// ---- 20_Product/20_ProBox/30_Toolbox/F_AssignTU_DataIndexToZone.TcPOU
FUNCTION F_AssignTU_DataIndexToZone : BOOL
(**************************************************************************************
 * 	Application		:	BoxControl Framework
 *	Revision		:	$Revision: $
 *	Revision date	:	$Date: $
 *	Last changed by	:	$Author: q8sheds $
 *	URL				:	$URL: $
 *
 *	Purpose			:	assign TU data to zone, overrides former method M_AssignTU_DataIndexToZone
 *
 * ------------------------------------------------------------------------------------
 *	Copyright Swisslog [IP AG], Switzerland. All rights reserved.
 * 
 * ------------------------------------------------------------------------------------
 *	
 * 	Revision History: 
 *
 * 	VERSION			DATE			INITIALS			DESCRIPTION
 *	0.1				2018-05-31		PkF/RtK					First Version
 *
 **************************************************************************************)
VAR_INPUT
	eFunctionNumber		: E_FunctionNumber;
	ZoneNumber			: INT; 
	TU_DataIndex		: DINT;
END_VAR

F_AssignTU_DataIndexToZone := FALSE;

// Check if function number and zone is valid
IF eFunctionNumber > E_FunctionNumber.F_BEGIN_FUNCTION AND
   eFunctionNumber < E_FunctionNumber.F_END_FUNCTION AND
   ZoneNumber > 0 AND ZoneNumber <= NUMBER_OF_ZONES_PER_FUNCTION THEN
  
   // yes, Zone number is valid	
	// Check reference is valid
    IF( NOT __ISVALIDREF(FunctionRegistry[eFunctionNumber].rFunction) OR
		NOT __ISVALIDREF(FunctionRegistry[eFunctionNumber].rSettingsFunction) OR
		NOT __ISVALIDREF(FunctionRegistry[eFunctionNumber].Zone[ZoneNumber].refZoneData)) THEN
		RETURN;  //bad references
	END_IF		
   
	
	IF ZoneNumber > 0 AND ZoneNumber <= FunctionRegistry[eFunctionNumber].rSettingsFunction.NumberOfZones THEN
		// TU Index is equal to the current
		IF TU_DataIndex > 0 AND FunctionRegistry[eFunctionNumber].Zone[ZoneNumber].refZoneData.TransportControlData.TU_DataIndex = 0 THEN
			// Assign TU data index						
			FunctionRegistry[eFunctionNumber].Zone[ZoneNumber].refZoneData.TransportControlData.TU_DataIndex := TU_DataIndex;
			//LastTU_DataIndex is not changed.
			FunctionRegistry[eFunctionNumber].Zone[ZoneNumber].refZoneData.TransportControlData.DataPresent := TRUE;
			F_AssignTU_DataIndexToZone := TRUE; 
		END_IF
	END_IF	   
      
END_IF

END_FUNCTION

// ---- 20_Product/20_ProBox/30_Toolbox/F_CheckAllFree.TcPOU
FUNCTION F_CheckAllFree : BOOL
(**************************************************************************************
 * 	Application		:	BoxControl Framework
 *	Revision		:	$Revision: 417092 $
 *	Revision date	:	$Date: 2018-11-14 12:58:58 +0100 (Mi., 14 Nov 2018) $
 *	Last changed by	:	$Author: q8aberh $
 *	URL				:	$URL: http://almscdc.swisslog.com/repo/SWPD/Development/ProMove/02_Controls/ProBox/03_Implementation/01_DevelopmentProject/01_Software/ProBox_COE/ProBox_DevProj_v1.0/PLC_1/20_Product/10_App/12_E_Functions/11_ProBox/02_Functions/02_TransportControl/F_Che $
 *
 *	Purpose			:	Return number of zones
 *
 * ------------------------------------------------------------------------------------
 *	Copyright Swisslog [IP AG], Switzerland. All rights reserved.
 * 
 * ------------------------------------------------------------------------------------
 *	
 * 	Revision History: 
 *
 * 	VERSION			DATE			INITIALS			DESCRIPTION
 *	0.1				01.01.2001		swl					Example
 *
 **************************************************************************************)
VAR_INPUT
	eFunctionNumber		: E_FunctionNumber; // Function number
END_VAR
VAR
	idx 				: INT; // Iterator
	AllFree				: BOOL; // Temp to check if all zones are occupied
END_VAR

// Check if function number is valid
IF eFunctionNumber > E_FunctionNumber.F_BEGIN_FUNCTION AND
   eFunctionNumber < E_FunctionNumber.F_END_FUNCTION THEN
  
   // Check reference is valid
   IF __ISVALIDREF(FunctionRegistry[eFunctionNumber].rSettingsFunction) THEN
		// Return All Free
		AllFree := TRUE;
		FOR idx := 1 TO FunctionRegistry[eFunctionNumber].rSettingsFunction.NumberOfZones DO
			IF FunctionRegistry[eFunctionNumber].Zone[idx].refZoneData.TransportControlData.Occupied THEN
				AllFree := FALSE;
				EXIT;
			END_IF
		END_FOR
		F_CheckAllFree := AllFree;
   END_IF
END_IF

END_FUNCTION

// ---- 20_Product/20_ProBox/30_Toolbox/F_CheckAllOccupied.TcPOU
FUNCTION F_CheckAllOccupied : BOOL
(**************************************************************************************
 * 	Application		:	BoxControl Framework
 *	Revision		:	$Revision: 417092 $
 *	Revision date	:	$Date: 2018-11-14 12:58:58 +0100 (Mi., 14 Nov 2018) $
 *	Last changed by	:	$Author: q8aberh $
 *	URL				:	$URL: http://almscdc.swisslog.com/repo/SWPD/Development/ProMove/02_Controls/ProBox/03_Implementation/01_DevelopmentProject/01_Software/ProBox_COE/ProBox_DevProj_v1.0/PLC_1/20_Product/10_App/12_E_Functions/11_ProBox/02_Functions/02_TransportControl/F_Che $
 *
 *	Purpose			:	Return number of zones
 *
 * ------------------------------------------------------------------------------------
 *	Copyright Swisslog [IP AG], Switzerland. All rights reserved.
 * 
 * ------------------------------------------------------------------------------------
 *	
 * 	Revision History: 
 *
 * 	VERSION			DATE			INITIALS			DESCRIPTION
 *	0.1				01.01.2001		swl					Example
 *
 **************************************************************************************)
VAR_INPUT
	eFunctionNumber		: E_FunctionNumber; // Function number
END_VAR
VAR
	idx 				: INT; // Iterator
	AllOccupied			: BOOL; // Temp to check if all zones are free
END_VAR

// Check if function number is valid
IF eFunctionNumber > E_FunctionNumber.F_BEGIN_FUNCTION AND
   eFunctionNumber < E_FunctionNumber.F_END_FUNCTION THEN
  
   // Check reference is valid
   IF __ISVALIDREF(FunctionRegistry[eFunctionNumber].rSettingsFunction) THEN
		// Return All Occupied
		AllOccupied := TRUE;
		FOR idx := 1 TO FunctionRegistry[eFunctionNumber].rSettingsFunction.NumberOfZones DO
			IF NOT FunctionRegistry[eFunctionNumber].Zone[idx].refZoneData.TransportControlData.Occupied THEN
				AllOccupied := FALSE;
				EXIT;
			END_IF
		END_FOR
		F_CheckAllOccupied := AllOccupied;
   END_IF
END_IF

END_FUNCTION

// ---- 20_Product/20_ProBox/30_Toolbox/F_CheckAllStarted.TcPOU
FUNCTION F_CheckAllStarted : BOOL
(**************************************************************************************
 * 	Application		:	BoxControl Framework
 *	Revision		:	$Revision: 417092 $
 *	Revision date	:	$Date: 2018-11-14 12:58:58 +0100 (Mi., 14 Nov 2018) $
 *	Last changed by	:	$Author: q8aberh $
 *	URL				:	$URL: http://almscdc.swisslog.com/repo/SWPD/Development/ProMove/02_Controls/ProBox/03_Implementation/01_DevelopmentProject/01_Software/ProBox_COE/ProBox_DevProj_v1.0/PLC_1/20_Product/10_App/12_E_Functions/11_ProBox/02_Functions/02_TransportControl/F_Che $
 *
 *	Purpose			:	Returns true if all the zones on the function are started
 *
 * ------------------------------------------------------------------------------------
 *	Copyright Swisslog [IP AG], Switzerland. All rights reserved.
 * 
 * ------------------------------------------------------------------------------------
 *	
 * 	Revision History: 
 *
 * 	VERSION			DATE			INITIALS			DESCRIPTION
 *	0.1				2018-08-14		PkF					First version
 *
 **************************************************************************************)
VAR_INPUT
	eFunctionNumber		: E_FunctionNumber; // Function number
END_VAR
VAR
	idx 				: INT; // Iterator
	AllStarted			: BOOL; // Temp to check if all zones are started
END_VAR

// Check if function number is valid
IF eFunctionNumber > E_FunctionNumber.F_BEGIN_FUNCTION AND
   eFunctionNumber < E_FunctionNumber.F_END_FUNCTION THEN
  
   // Check reference is valid
   IF __ISVALIDREF(FunctionRegistry[eFunctionNumber].rSettingsFunction) AND 
		__ISVALIDREF(FunctionRegistry[eFunctionNumber].rFunctionData) THEN
		// Return All Started
		AllStarted := TRUE;
		FOR idx := 1 TO FunctionRegistry[eFunctionNumber].rSettingsFunction.NumberOfZones DO
			IF (FunctionRegistry[eFunctionNumber].rFunctionData.OperationState.eState <> E_PositionState.STARTED AND 
				FunctionRegistry[eFunctionNumber].rFunctionData.OperationState.eState <> E_PositionState.STOPPING) OR 
				FunctionRegistry[eFunctionNumber].rFunctionData.ErrorData.ZoneErrorPending THEN
				AllStarted := FALSE;
				EXIT;
			END_IF
		END_FOR
		F_CheckAllStarted := AllStarted;
   END_IF
END_IF

END_FUNCTION

// ---- 20_Product/20_ProBox/30_Toolbox/F_DeleteTU_DataIndex.TcPOU
FUNCTION F_DeleteTU_DataIndex : BOOL
(**************************************************************************************
 * 	Application		:	BoxControl Framework
 *	Revision		:	$Revision: 417092 $
 *	Revision date	:	$Date: 2018-11-14 12:58:58 +0100 (Mi., 14 Nov 2018) $
 *	Last changed by	:	$Author: q8aberh $
 *	URL				:	$URL: http://almscdc.swisslog.com/repo/SWPD/Development/ProMove/02_Controls/ProBox/03_Implementation/01_DevelopmentProject/01_Software/ProBox_COE/ProBox_DevProj_v1.0/PLC_1/20_Product/10_App/12_E_Functions/11_ProBox/02_Functions/F_DeleteTU_DataIndex.TcPO $
 *
 *	Purpose			:	Moves TU data from a position.
 *
 * ------------------------------------------------------------------------------------
 *	Copyright Swisslog [IP AG], Switzerland. All rights reserved.
 * 
 * ------------------------------------------------------------------------------------
 *	
 * 	Revision History: 
 *
 * 	VERSION			DATE			INITIALS			DESCRIPTION
 *	0.1				01.01.2001		swl					Example
 *
 **************************************************************************************)
VAR_INPUT
	eFunctionNumber	: E_FunctionNumber; // Function number of corresponding function
	mZoneNumber 	: INT; // Zone number
END_VAR

VAR
	STI_Instance	: ITF_SubsystemTransport; // Instance to compare valid interfaces
END_VAR

// Check if function number is valid
IF eFunctionNumber > E_FunctionNumber.F_BEGIN_FUNCTION AND
   eFunctionNumber < E_FunctionNumber.F_END_FUNCTION THEN
  
	// Check reference is valid
	IF __ISVALIDREF(FunctionRegistry[eFunctionNumber].rFunction) THEN
   		// Return tu data index
   		F_DeleteTU_DataIndex := FunctionRegistry[eFunctionNumber].rFunction.M_DeleteTU_DataIndex(
						mZoneNumber := mZoneNumber,
						mTU_DataIndex := F_GetTU_DataIndex(
												eFunctionNumber := eFunctionNumber,
												ZoneNumber := mZoneNumber),
						mInit	:= FALSE);
	END_IF
END_IF

END_FUNCTION

// ---- 20_Product/20_ProBox/30_Toolbox/F_PB_GetTransportData.TcPOU
FUNCTION F_PB_GetTransportData : ST_TransportData
(**************************************************************************************
 * 	Application		:	BoxControl Framework
 *	Revision		:	$Revision:  $
 *	Revision date	:	$Date: $
 *	Last changed by	:	$Author: q8sheds $
 *	URL				:	$URL: $
 *
 *	Purpose			:	return Transport data
 *
 * ------------------------------------------------------------------------------------
 *	Copyright Swisslog [IP AG], Switzerland. All rights reserved.
 * 
 * ------------------------------------------------------------------------------------
 *	
 * 	Revision History: 
 *
 * 	VERSION			DATE			INITIALS			DESCRIPTION
 *	0.1				01.01.2001		swl					Example
 *
 **************************************************************************************)
VAR_INPUT
	eFunctionNumber		: E_FunctionNumber; // Function number
	ZoneNumber			: INT; // Zone number
END_VAR



VAR
	FunctionBase: INT;
END_VAR


//init default data
F_PB_GetTransportData.eFunctionNumber := E_FunctionNumber.F_BEGIN_FUNCTION;
F_PB_GetTransportData.ZoneNumber:=0;
F_PB_GetTransportData.rTransportControlData REF= PBTransportCtrl.pbTransportControlDataEmpty;
F_PB_GetTransportData.rSettings REF= PBTransportCtrl.pbZoneSettingsEmpty;


// Check if function number is valid
IF eFunctionNumber > E_FunctionNumber.F_BEGIN_FUNCTION AND
   eFunctionNumber < E_FunctionNumber.F_END_FUNCTION AND
   ZoneNumber > 0 AND ZoneNumber <= NUMBER_OF_ZONES_PER_FUNCTION THEN
  
	// Check reference is valid
	IF __ISVALIDREF(FunctionRegistry[eFunctionNumber].Zone[ZoneNumber].refZoneData) THEN
   		// Set transport data
   		//F_PB_GetTransportControlDataRef REF= FunctionRegistry[eFunctionNumber].Zone[ZoneNumber].refZoneData.TransportControlData;
		F_PB_GetTransportData.eFunctionNumber := eFunctionNumber;
		F_PB_GetTransportData.ZoneNumber := ZoneNumber;
		F_PB_GetTransportData.rSettings REF= FunctionRegistry[eFunctionNumber].rSettingsFunction.Zone[ZoneNumber];
		F_PB_GetTransportData.rTransportControlData REF= FunctionRegistry[eFunctionNumber].Zone[ZoneNumber].refZoneData.TransportControlData;				
	END_IF
END_IF

END_FUNCTION

// ---- 20_Product/20_ProBox/30_Toolbox/F_PB_GetZoneITC.TcPOU
FUNCTION F_PB_GetZoneITC : ST_ITC_Zone
VAR_INPUT
		eFunctionNumber		: E_FunctionNumber; // Function number
		ZoneNumber			: INT := 1;
END_VAR
VAR
END_VAR

// Check if function number is validas
IF eFunctionNumber > E_FunctionNumber.F_BEGIN_FUNCTION AND
   eFunctionNumber < E_FunctionNumber.F_END_FUNCTION THEN
  
	// Check reference is valid
	IF __ISVALIDREF(FunctionRegistry[eFunctionNumber].rFunctionInterface) THEN
   		// Return function interlock
   		F_PB_GetZoneITC := FunctionRegistry[eFunctionNumber].rFunction.ITC.ZoneITC[ZoneNumber];
	END_IF
END_IF

END_FUNCTION

// ---- 20_Product/20_ProBox/30_Toolbox/F_PB_IsLogicalOccupied.TcPOU
//A zone is occupied until the TU is handed over completly, or when the takeover is fully completed
FUNCTION F_PB_IsLogicalOccupied : BOOL
VAR_INPUT
	TransportControlData : REFERENCE TO ST_TransportControlData;
END_VAR
VAR
END_VAR


IF(NOT __ISVALIDREF(TransportControlData)) THEN RETURN; END_IF;

F_PB_IsLogicalOccupied := TransportControlData.Occupied OR TransportControlData.eTransportState = E_TransportState.HANDOVER;

END_FUNCTION

// ---- 20_Product/20_ProBox/30_Toolbox/F_PB_SetDestination.TcPOU
//Set destination to an already existing TU Table dataset
FUNCTION F_PB_SetDestination : BOOL
(**************************************************************************************
 * 	Application		:	ProBox
 *	Revision		:	$$
 *	Revision date	:	$$
 *	Last changed by	:	$$
 *	URL				:	$$
 *
 *	Purpose			:	Set a destination to an existing TU Table dataset.
 * 						Remark: as Tu_Table is persistant memory type, one should not repeatedly write to the TU_Table 
 *
 * ------------------------------------------------------------------------------------
 *	Copyright Swisslog [IP AG], Switzerland. All rights reserved.  
 **************************************************************************************)
VAR_INPUT
	TuDataIndex			: DINT; // Existing TU data table index there the Destination shall be assigned to
	Destination			: E_FunctionNumber; // Destination function
	DestinationZone		: INT:=1; // Destination zone
	ForceOverwrite		: BOOL:=FALSE; //Set to true in order to overwrite an existing valid destination and to be sure only writing once.
	AssignTuType		: BOOL:=FALSE; //Set to true to assign TuType
	TuType				: INT:=0;
	InsertFunction		: E_FunctionNumber:= E_FunctionNumber.F_BEGIN_FUNCTION;	//Optional data that is written to TimeStamp 
	InsertZone			: INT:=0;		
END_VAR
VAR
	DataSetDestIndex	: INT:=1;
END_VAR

//Sanity check
IF( TuDataIndex<=0 OR TuDataIndex>Conveyor.NUMBER_OF_TU_DATA OR
	Destination<= E_FunctionNumber.F_BEGIN_FUNCTION OR Destination>= E_FunctionNumber.F_END_FUNCTION OR
	DestinationZone <=0 OR DestinationZone > Conveyor.NUMBER_OF_ZONES_PER_FUNCTION) THEN
	RETURN; //invalid arguments
END_IF

IF(ForceOverwrite = FALSE AND TU_DataTable[TuDataIndex].DataSet.JobPresent) THEN
	RETURN; //JobPresent is active, so dont overwrite data again..
END_IF 


// Update TU Data set
TU_DataTable[TuDataIndex].DataSet.DataPresent:= TRUE;
TU_DataTable[TuDataIndex].DataSet.NumberOfDest	:= 1;				
TU_DataTable[TuDataIndex].DataSet.JobPresent := Destination > E_FunctionNumber.F_BEGIN_FUNCTION AND Destination<>InsertFunction;
TU_DataTable[TuDataIndex].Destination[DataSetDestIndex].eFunctionNumber := Destination;
TU_DataTable[TuDataIndex].Destination[DataSetDestIndex].ZoneNumber := DestinationZone;
TU_DataTable[TuDataIndex].Destination[DataSetDestIndex].PositionName := FunctionRegistry[Destination].FunctionName;

//Update TimeStamp
TU_DataTable[TuDataIndex].TimeStamp.eInsertFunctionNumber := InsertFunction;
TU_DataTable[TuDataIndex].TimeStamp.InsertZoneNumber:=InsertZone;
TU_DataTable[TuDataIndex].TimeStamp.InsertDateTime := System.fbSystemTime.TIMESTR;

//Set TU_Type?
IF(AssignTuType) THEN
	TU_DataTable[TuDataIndex].DataSet.TU_Type := TuType;
END_IF;


F_PB_SetDestination := TRUE;

END_FUNCTION

// ---- 20_Product/20_ProBox/30_Toolbox/F_PB_SetPalletOrientation.TcPOU
//Rotate profile data 90,80 or 270 degrees
FUNCTION F_PB_SetPalletOrientation : BOOL
VAR_INPUT
	ePalletOrientation  : E_PalletOrientation;	
	TuTableIdx			: DINT; // Which Tu Table destination slot (Default 1)
END_VAR
VAR
	TU_DataIndex  : DINT;
	_ProfileData: ST_Profile;
	_TempProfileData : ST_Profile;
	InvertedDone : BOOL:= FALSE;
END_VAR

//Sanity check
IF TuTableIdx <= 0 OR ePalletOrientation = OrientationZero THEN	
	RETURN;
END_IF

TU_DataIndex := TuTableIdx;
_ProfileData:= TU_DataTable[TU_DataIndex].Profile;	


CASE ePalletOrientation OF 	
	OrientationZero:
		; //nothing to do	

	OrientationNinty:
		TU_DataTable[TU_DataIndex].Profile.ProfileLeft:= _ProfileData.ProfileRear;	
		TU_DataTable[TU_DataIndex].Profile.ProfileRight:= _ProfileData.ProfileFront;	
		TU_DataTable[TU_DataIndex].Profile.ProfileFront:= _ProfileData.ProfileLeft;
		TU_DataTable[TU_DataIndex].Profile.ProfileRear:= _ProfileData.ProfileRight;
	
	OrientationOneEighty:
		TU_DataTable[TU_DataIndex].Profile.ProfileLeft:= _ProfileData.ProfileRight;
		TU_DataTable[TU_DataIndex].Profile.ProfileRight:= _ProfileData.ProfileLeft;
		TU_DataTable[TU_DataIndex].Profile.ProfileFront:= _ProfileData.ProfileRear;
		TU_DataTable[TU_DataIndex].Profile.ProfileRear:= _ProfileData.ProfileFront;
	
	OrientationTwoSeventy:
		TU_DataTable[TU_DataIndex].Profile.ProfileLeft:= _ProfileData.ProfileFront;
		TU_DataTable[TU_DataIndex].Profile.ProfileRight:= _ProfileData.ProfileRear;
		TU_DataTable[TU_DataIndex].Profile.ProfileFront:= _ProfileData.ProfileRight;
		TU_DataTable[TU_DataIndex].Profile.ProfileRear:= _ProfileData.ProfileLeft;
END_CASE

F_PB_SetPalletOrientation:=TRUE; ;

END_FUNCTION

// ---- 20_Product/20_ProBox/30_Toolbox/F_SetOccupied.TcPOU
FUNCTION F_SetOccupied : BOOL
(**************************************************************************************
 * 	Application		:	BoxControl Framework
 *	Revision		:	$Revision: 417092 $
 *	Revision date	:	$Date: 2018-11-14 12:58:58 +0100 (Mi., 14 Nov 2018) $
 *	Last changed by	:	$Author: q8aberh $
 *	URL				:	$URL: http://almscdc.swisslog.com/repo/SWPD/Development/ProMove/02_Controls/ProBox/03_Implementation/01_DevelopmentProject/01_Software/ProBox_COE/ProBox_DevProj_v1.0/PLC_1/20_Product/10_App/12_E_Functions/11_ProBox/02_Functions/F_SetOccupied.TcPOU $
 *
 *	Purpose			:	Return zone data
 *
 * ------------------------------------------------------------------------------------
 *	Copyright Swisslog [IP AG], Switzerland. All rights reserved.
 * 
 * ------------------------------------------------------------------------------------
 *	
 * 	Revision History: 
 *
 * 	VERSION			DATE			INITIALS			DESCRIPTION
 *	0.1				01.01.2001		swl					Example
 *
 **************************************************************************************)
VAR_INPUT
	eFunctionNumber		: E_FunctionNumber;
	ZoneNumber			: INT; 
END_VAR



// Check if function number and zone is valid
IF eFunctionNumber > E_FunctionNumber.F_BEGIN_FUNCTION AND
   eFunctionNumber < E_FunctionNumber.F_END_FUNCTION AND
   ZoneNumber > 0 AND ZoneNumber <= NUMBER_OF_ZONES_PER_FUNCTION THEN
  
	// Check reference is valid
    IF __ISVALIDREF(FunctionRegistry[eFunctionNumber].rFunction) THEN
	   // Return zone data
		IF __ISVALIDREF(FunctionRegistry[eFunctionNumber].Zone[ZoneNumber].refZoneData) THEN
			FunctionRegistry[eFunctionNumber].Zone[ZoneNumber].refZoneData.TransportControlData.Occupied := TRUE;
			FunctionRegistry[eFunctionNumber].Zone[ZoneNumber].refZoneData.TransportControlData.NumberOfPresentTUs :=1;
			FunctionRegistry[eFunctionNumber].Zone[ZoneNumber].refZoneData.TransportControlData.eTransportState := E_TransportState.OCCUPIED;
			F_SetOccupied:=TRUE;
	   END_IF
	    	   
    END_IF  
END_IF

END_FUNCTION

// ---- 20_Product/20_ProBox/40_TC_Visualization/99_SIS/FB_VizuSIS.TcPOU
FUNCTION_BLOCK FB_VizuSIS
VAR_INPUT
	ATQ				: BOOL;
	RTQ				: BOOL;
	TTA				: BOOL;
	TDQ				: BOOL;
	TTA_Destination	: STRING(NAME_LENGTH) := '10-001-0100-01-1';
	PositionString	: STRING(NAME_LENGTH) := '10-001-0100-01-1'; // Name of position 11-111-1111-11-1;	
	ATQ_Dimension	: ST_Dimension :=(Width:=800, Length:=800, Height:=500, Weight:=1200);
	ATQ_Label		: STRING(Conveyor.LABEL_LENGTH) := 'CREATECODE';
	TU_ID			: STRING(Conveyor.TU_ID_STRINGLENGTH):= Conveyor.TU_ID_UNKNOWN; // TU-ID
	AssignmentID	: UDINT := Conveyor.ASSIGNMENT_ID_UNKNOWN;
	AutoID			: BOOL; //Use TU ID and Assignment ID from TU table for TTA and TDQ
END_VAR
VAR_OUTPUT
	BadPosition		: BOOL;
END_VAR
VAR
	myPos			: STRING(NAME_LENGTH);
	myTuIndex		: DINT;

	TrigATQ : R_TRIG();
	TrigRTQ : R_TRIG();
	TrigTTA : R_TRIG();
	TrigTDQ : R_TRIG();
	
END_VAR
VAR_TEMP
	Position : ST_PositionIdent;
END_VAR

myPos := F_ReduceToAlphaNumeric(PositionString);
Position := F_SearchFunctionPosition(Position := myPos);
BadPosition := Position.eFunctionNumber = E_FunctionNumber.F_BEGIN_FUNCTION;
IF(BadPosition) THEN
	RETURN;
END_IF


TrigATQ(CLK:=ATQ);
TrigRTQ(CLK:=RTQ);
TrigTTA(CLK:=TTA);
TrigTDQ(CLK:=TDQ);

IF(TrigATQ.Q) THEN
	//ATQDimension
	_M_SendATQ(Position,ATQ_Dimension,ATQ_Label);
	//F_AddPhysicalTU(Position.eFunctionNumber,Position.ZoneNumber);
END_IF

IF(TrigRTQ.Q) THEN
	F_RemovePhysicalTU(Position.eFunctionNumber,Position.ZoneNumber);
END_IF

IF(TrigTTA.Q) THEN	
	_M_SendTTA(Position,TTA_Destination,TU_ID,AssignmentID);
END_IF

IF(TrigTDQ.Q) THEN	
	_M_SendTDQ(Position);
END_IF

METHOD PRIVATE _M_GetIDs : BOOL
VAR_INPUT
	Position 		: REFERENCE TO ST_PositionIdent;	
	TU_ID			: REFERENCE TO STRING(Conveyor.TU_ID_STRINGLENGTH); // TU-ID
	AssigID			: REFERENCE TO UDINT ;
END_VAR

VAR
	myTuIndex		: DINT;
END_VAR
//(Conveyor.TU_ID_STRINGLENGTH):= Conveyor.TU_ID_UNKNOWN;
//:= Conveyor.ASSIGNMENT_ID_UNKNOWN

IF(THIS^.AutoID) THEN
	
	myTuIndex := F_PB_GetTransportControlDataRef(Position.eFunctionNumber,Position.ZoneNumber).TU_DataIndex;
	IF(myTuIndex>0) THEN
		AssigID		:= TU_Table.TU_DataTable[myTuIndex].AssignmentID;
		TU_ID 			:= TU_Table.TU_DataTable[myTuIndex].TU_ID.ASCII;
	ELSE
		AssigID 		:= Conveyor.ASSIGNMENT_ID_UNKNOWN;
		TU_ID		:= Conveyor.TU_ID_UNKNOWN;	
	END_IF	
ELSE
	//use the ID's from the input field of the vizio interface.
	TU_ID := THIS^.TU_ID;	
	AssigID := THIS^.AssignmentID;
END_IF
END_METHOD

METHOD PRIVATE _M_SendATQ : BOOL
VAR_INPUT
	Position 		: REFERENCE TO ST_PositionIdent;
	Dimension		: REFERENCE TO ST_Dimension;
	Label			: REFERENCE TO STRING(Conveyor.LABEL_LENGTH);	
END_VAR
VAR
	myLabel			: STRING(Conveyor.LABEL_LENGTH);
END_VAR
VAR_STAT
	ID		: INT := 1;
	ATQ		: ST_ITC_ATQ;
END_VAR

ATQ.Position := F_ReduceToAlphaNumeric(InputString := Position.PositionName);

IF(Label[0]=0) THEN

	myLabel := F_StuffString(
			InputString 	:= INT_TO_STRING(ID), 
			StringLength	:= 8, 
			StuffCharacter 	:= '0',
			LeftAligned     := FALSE);
	myLabel := CONCAT('TESTLABEL_',myLabel);
			
	ID := ID + 1;
	IF ID > 9998 THEN
		ID := 1;
	END_IF
ELSE
	myLabel := Label;
END_IF		

IF(Dimension.Height=0) THEN Dimension.Height:=200; END_IF
IF(Dimension.Length=0) THEN Dimension.Length:=200; END_IF
IF(Dimension.Weight=0) THEN Dimension.Weight:=200; END_IF
IF(Dimension.Width=0) THEN Dimension.Width:=200; END_IF

ATQ.Height := Dimension.Height;
ATQ.Length := Dimension.Length;
ATQ.Weight := Dimension.Weight;
ATQ.Width := Dimension.Width;

ATQ.LabelPresent := 1;
ATQ.Label := myLabel;


IF(ProBoxSystem.EMULATION_ENABLED) THEN
	fbITC_ManagerEmulation.M_AddData(
		meChannelSrc := 0,
		mMsgType     := E_ITC_MsgTypeConv.E_ADD_TU_REQUEST,
		mpData		 := ADR(ATQ),
		mLen 		 := SIZEOF(ATQ));
END_IF
END_METHOD

METHOD PRIVATE _M_SendTDQ : BOOL
VAR_INPUT
	Position 		: REFERENCE TO ST_PositionIdent;	
	//TU_Id    		: STRING(Conveyor.TU_ID_STRINGLENGTH);
END_VAR
VAR	
	TDQ		: ST_ITC_TDQ;
	
END_VAR

_M_GetIDs(Position,TDQ.TU_ID, TDQ.AssignmentID);

TDQ.Position := F_ReduceToAlphaNumeric(InputString := Position.PositionName);

TDQ.Code :=0;
TDQ.MsgSequence:=999;


_M_SendTDQ:= fbITC_Manager.M_AddData(
					meChannelSrc := 0,
					mMsgType     := E_ITC_MsgTypeConv.TASK_DELETE_REQUEST,
					mpData		 := ADR(TDQ),
					mLen		 := SIZEOF(TDQ));
END_METHOD

METHOD PRIVATE _M_SendTTA : BOOL
VAR_INPUT
	Position 		: REFERENCE TO ST_PositionIdent;
	Destination		: REFERENCE TO STRING(NAME_LENGTH);
	TU_Id    		: STRING(Conveyor.TU_ID_STRINGLENGTH);
	AssignmentID	: UDINT := Conveyor.ASSIGNMENT_ID_UNKNOWN;
END_VAR
VAR
	TTA		: ST_ITC_TTA;
	//mName	: STRING[NAME_LENGTH];
END_VAR
//mName := F_GetFunctionName(eFunctionNumber:= Position.eFunctionNumber, ZoneNumber:= Position.ZoneNumber);
TTA.Position := F_ReduceToAlphaNumeric(InputString := Position.PositionName);
//mName := F_GetFunctionName(eFunctionNumber:= Position.eFunctionNumber, ZoneNumber:= Position.ZoneNumber);
TTA.Destination[1] := F_ReduceToAlphaNumeric(InputString := Destination);//'11-001-0206-01-1';
TTA.DestinationSlot:=1;
TTA.NumberOfDestinations:=1;
TTA.AssignmentID:=AssignmentID;
TTA.TU_ID := TU_Id;

_M_GetIDs(Position,TTA.TU_ID, TTA.AssignmentID);

_M_SendTTA:= fbITC_Manager.M_AddData(
					meChannelSrc := 0,
					mMsgType     := E_ITC_MsgTypeConv.TRANSPORT_TASK_ASSIGNMENT,
					mpData		 := ADR(TTA),
					mLen		 := SIZEOF(TTA));
END_METHOD

END_FUNCTION_BLOCK

// ---- 20_Product/30_Toolbox/12_StringStream/F_CompareAlphaNumericString.TcPOU
FUNCTION F_CompareAlphaNumericString : BOOL
(**************************************************************************************
 * 	Application		:	BoxControl Framework
 *	Revision		:	$Revision: 404529 $
 *	Revision date	:	$Date: 2018-04-23 08:21:38 +0200 (Mo., 23 Apr 2018) $
 *	Last changed by	:	$Author: b7bolm $
 *	URL				:	$URL: http://almscdc.swisslog.com/repo/SWPD/Development/BoxControlFramework/20_Release/trunk/01_Software/BCF/BCF/JumpStart/30_Toolbox/12_StringStream/F_CompareAlphaNumericString.TcPOU $
 *
 *	Purpose			:	Compares two strings. Chars which are not from the 
 *						following type are ignored: 0..9, A..Z, a..z.
 *						Example: 21-001-0010-001 -> 210010010001
 *						Return value will be TRUE if both strings are identical.
 *						
 *						Length allows to compare only a certain part of a string.
 *
 * ------------------------------------------------------------------------------------
 *	Copyright Swisslog [IP AG], Switzerland. All rights reserved.
 * 
 * ------------------------------------------------------------------------------------
 *	
 * 	Revision History: 
 *
 * 	VERSION			DATE			INITIALS			DESCRIPTION
 *	0.1				01.01.2001		swl					Example
 *
 **************************************************************************************)
VAR_INPUT
	InputString1		: STRING(100); // Compare string 1
	InputString2		: STRING(100); // Compare string 2
	Length				: INT; // Length of input string
END_VAR

VAR
	pASCII_ARRAY_1  	: POINTER TO ARRAY [1..100] OF BYTE; // Pointer for mapping 
	ASCII_Value_1		: INT; // Value of the ascii-cahr 
	pASCII_ARRAY_2  	: POINTER TO ARRAY [1..100] OF BYTE; // Pointer for mapping 
	ASCII_Value_2		: INT; // Value of the ascii-cahr 
	Idx 				: INT; // Index variable 
	ArrayIdx_1			: INT; // Index variable 
	ArrayIdx_2			: INT; // Index variable 
	ASCII_OK_1			: BOOL; // Char is a alphanumeric sign 
	ASCII_OK_2			: BOOL; // Char is a alphanumeric sign 
END_VAR

// Initialize
F_CompareAlphaNumericString := FALSE;
ArrayIdx_1 := 1;
ArrayIdx_2 := 1;

// Create pointer of the InputString 
pASCII_ARRAY_1 := ADR(InputString1);
pASCII_ARRAY_2 := ADR(InputString2);

// Go trough strings
FOR Idx := 1 TO Length DO
	// Get first sign
	ASCII_Value_1 := BYTE_TO_INT(pASCII_ARRAY_1^[ArrayIdx_1]);
	
	// Only if it is a char between 0..9, A..Z, a..z 
	ASCII_OK_1 := ((ASCII_Value_1 > 47) AND (ASCII_Value_1 < 58))
		 	OR ((ASCII_Value_1 > 64) AND (ASCII_Value_1 < 91))
			OR ((ASCII_Value_1 > 96) AND (ASCII_Value_1 < 123));

	// Get second sign
	ASCII_Value_2 := BYTE_TO_INT(pASCII_ARRAY_2^[ArrayIdx_2]);
	
	// Only if it is a char between 0..9, A..Z, a..z 
	ASCII_OK_2 := ((ASCII_Value_2 > 47) AND (ASCII_Value_2 < 58))
			OR ((ASCII_Value_2 > 64) AND (ASCII_Value_2 < 91))
			OR ((ASCII_Value_2 > 96) AND (ASCII_Value_2 < 123));

	// Both chars are alphanumeric 
	IF ASCII_OK_1 AND ASCII_OK_2 THEN
		// Both are the same
		IF ASCII_Value_1 = ASCII_Value_2 THEN
			// Continue
			F_CompareAlphaNumericString := TRUE;
			// Increment index
			ArrayIdx_1 := ArrayIdx_1 + 1;
			ArrayIdx_2 := ArrayIdx_2 + 1;
		ELSE
			// Not equal - stop
			F_CompareAlphaNumericString := FALSE;
			RETURN;
		END_IF
	// Char of string 1 is not alphanumeric, jump to the next char of string 1 
	ELSIF NOT ASCII_OK_1 AND ASCII_OK_2 THEN
		ArrayIdx_1 := ArrayIdx_1 + 1;

	// Char of string 2 is not alphanumeric, jump to the next char of string 2 
	ELSIF ASCII_OK_1 AND NOT ASCII_OK_2 THEN
		ArrayIdx_2 := ArrayIdx_2 + 1;

	// Char of string 1 and 2 are not alphanumeric, jump to the next char of both strings 
	ELSE
		ArrayIdx_1 := ArrayIdx_1 + 1;
		ArrayIdx_2 := ArrayIdx_2 + 1;
	END_IF
END_FOR

END_FUNCTION

// ---- 20_Product/30_Toolbox/12_StringStream/F_MaxReportTime_TO_Time.TcPOU
FUNCTION F_MaxReportTime_TO_Time : TIME
VAR_INPUT
	sTimeIn : STRING;
END_VAR
VAR
	TempOT : OTSTRUCT;
	
	
END_VAR

//'12:34:56:789';
TempOT.wHour			:= STRING_TO_WORD(LEFT(sTimeIn,2));
TempOT.wMinute			:= STRING_TO_WORD(MID(sTimeIn,2,4));
TempOT.wSecond			:= STRING_TO_WORD(MID(sTimeIn,2,7));

F_MaxReportTime_TO_Time	:= OTSTRUCT_TO_TIME(OTIN:= TempOT);

END_FUNCTION

// ---- 20_Product/30_Toolbox/12_StringStream/F_RemoveSign.TcPOU
FUNCTION F_RemoveSign : STRING(255)
(**************************************************************************************
 * 	Application		:	BoxControl Framework
 *	Revision		:	$Revision: 404529 $
 *	Revision date	:	$Date: 2018-04-23 08:21:38 +0200 (Mo., 23 Apr 2018) $
 *	Last changed by	:	$Author: b7bolm $
 *	URL				:	$URL: http://almscdc.swisslog.com/repo/SWPD/Development/BoxControlFramework/20_Release/trunk/01_Software/BCF/BCF/JumpStart/30_Toolbox/12_StringStream/F_RemoveSign.TcPOU $
 *
 *	Purpose			:	Remove a sign from a string.
 *
 * ------------------------------------------------------------------------------------
 *	Copyright Swisslog [IP AG], Switzerland. All rights reserved.
 * 
 * ------------------------------------------------------------------------------------
 *	
 * 	Revision History: 
 *
 * 	VERSION			DATE			INITIALS			DESCRIPTION
 *	0.1				01.01.2001		swl					Example
 *
 **************************************************************************************)
VAR_INPUT
	InputString		: STRING(255); // Input string
	Sign			: STRING(1); // Sign to remove
END_VAR
VAR
	Idx				: INT; // Iterator
	pASCII_Array	: POINTER TO ARRAY[1..255] OF BYTE;
	pSign			: POINTER TO BYTE;
	ASCII_Value		: INT; // Value
END_VAR

// Initialize
F_RemoveSign := '';

// Build ASCII array and sign as byte
pASCII_Array := ADR(InputString);
pSign := ADR(Sign);

// Go Through string
FOR Idx := 1 TO LEN(InputString) DO
	// Get first ASCII sign as INT
	ASCII_Value := BYTE_TO_INT(pASCII_Array^[Idx]);
	
	// Add all except sign to new string
	IF pSign^ <> ASCII_Value THEN
		// Build string
		fbFormatString( sFormat := '%C',
						arg1 	:= F_BYTE(pASCII_Array^[Idx]));
		
		// Return alpha numeric string
		F_RemoveSign := CONCAT(F_RemoveSign, fbFormatString.sOut);
	END_IF
END_FOR

END_FUNCTION

// ---- 20_Product/30_Toolbox/12_StringStream/F_SampleTime_TO_TIME.TcPOU
FUNCTION F_SampleTime_TO_TIME : TIME
VAR_INPUT
	SampleTimeString : STRING;
END_VAR
VAR
	TempOT : OTSTRUCT;
	
	
END_VAR

//'12:34:56:789';


TempOT.wHour			:= STRING_TO_WORD(LEFT(SampleTimeString,2));
TempOT.wMinute			:= STRING_TO_WORD(MID(SampleTimeString,2,4));
TempOT.wSecond			:= STRING_TO_WORD(MID(SampleTimeString,2,7));
TempOT.wMilliseconds	:= STRING_TO_WORD(RIGHT(SampleTimeString,3));


F_SampleTime_TO_TIME:= OTSTRUCT_TO_TIME(TempOT);

END_FUNCTION

// ---- 20_Product/30_Toolbox/12_StringStream/F_Time_TO_MaxReportTime.TcPOU
FUNCTION F_Time_TO_MaxReportTime : STRING
VAR_INPUT
	TIN: TIME;
END_VAR
VAR
	TempOT	:OTSTRUCT;
	TempHr	:STRING(2);
	TempMinute	:STRING(2);
	TempSecond	:STRING(2);

END_VAR

	
TempOT:= TIME_TO_OTSTRUCT(TIN:=TIN );
TempHr:= F_StuffString(InputString := WORD_TO_STRING(TempOT.wHour),StringLength	:= 2,StuffCharacter:= '0',LeftAligned := FALSE);
TempMinute:= F_StuffString(InputString := WORD_TO_STRING(TempOT.wMinute),StringLength	:= 2,StuffCharacter:= '0',LeftAligned := FALSE);
TempSecond:= F_StuffString(InputString := WORD_TO_STRING(TempOT.wSecond),StringLength	:= 2,StuffCharacter:= '0', LeftAligned := FALSE);


F_Time_TO_MaxReportTime:= CONCAT(F_Time_TO_MaxReportTime,TempHr);
F_Time_TO_MaxReportTime:= CONCAT(F_Time_TO_MaxReportTime,':');
F_Time_TO_MaxReportTime:= CONCAT(F_Time_TO_MaxReportTime,TempMinute);
F_Time_TO_MaxReportTime:= CONCAT(F_Time_TO_MaxReportTime,':');
F_Time_TO_MaxReportTime:= CONCAT(F_Time_TO_MaxReportTime,TempSecond);

END_FUNCTION

// ---- 20_Product/30_Toolbox/12_StringStream/F_Time_TO_SampleTime.TcPOU
FUNCTION F_Time_TO_SampleTime : STRING
VAR_INPUT
	TIN: TIME;
END_VAR
VAR
	TempOT		:OTSTRUCT;
	TempHour	:STRING(2);
	TempMinute	:STRING(2);
	TempSecond	:STRING(2);
	TempMillisecond	:STRING(3);	
END_VAR

	
TempOT:= TIME_TO_OTSTRUCT(TIN:=TIN );

TempHour 		:= F_StuffString(InputString:= WORD_TO_STRING(TempOT.wHour), StringLength	:= 2,StuffCharacter 	:= '0', LeftAligned := FALSE);
TempMinute 		:= F_StuffString(InputString:= WORD_TO_STRING(TempOT.wMinute), StringLength	:= 2,StuffCharacter 	:= '0', LeftAligned := FALSE);
TempSecond 		:= F_StuffString(InputString:= WORD_TO_STRING(TempOT.wSecond), StringLength	:= 2,StuffCharacter 	:= '0', LeftAligned := FALSE);
TempMillisecond := F_StuffString(InputString:= WORD_TO_STRING(TempOT.wMilliseconds), StringLength	:= 3,StuffCharacter 	:= '0', LeftAligned := FALSE);

F_Time_TO_SampleTime:= CONCAT(F_Time_TO_SampleTime,TempHour);
F_Time_TO_SampleTime:= CONCAT(F_Time_TO_SampleTime,':');
F_Time_TO_SampleTime:= CONCAT(F_Time_TO_SampleTime,TempMinute);
F_Time_TO_SampleTime:= CONCAT(F_Time_TO_SampleTime,':');
F_Time_TO_SampleTime:= CONCAT(F_Time_TO_SampleTime,TempSecond);
F_Time_TO_SampleTime:= CONCAT(F_Time_TO_SampleTime,'.');
F_Time_TO_SampleTime:= CONCAT(F_Time_TO_SampleTime,TempMillisecond);

END_FUNCTION

// ---- 20_Product/30_Toolbox/16_Sequencing/10_Core/FB_SeqBranch.TcPOU
/// Function block is able to decide if a waiting TU is allowed to move, 
/// considering one branch.
FUNCTION_BLOCK FB_SeqBranch
(************************************************************************************** 
* 	Application 		: BoxControl Framework 
* 	Revision 			: $Revision: 404877 $ 
* 	Revision date 		: $Date: 2018-04-26 14:10:34 +0200 (Thu, 26 Apr 2018) $ 
* 	Last changed by 	: $Author: b7ernsb $ 
* 	URL 				: $URL: http://almscdc.swisslog.com/repo/SWPD/Development/BoxControlFramework/21_Projects/BCF_2.0/trunk/BCF/BCF/JumpStart/20_Product/10_App/12_E_Functions/10_Lib/10_Conv/FB_FunctionConv.TcPOU $ 
* ------------------------------------------------------------------------------------ 
* 	© Swisslog AG 
* 	Swisslog is not liable for any usage of this source code that is not agreed 
* 	on between Swisslog and the other party. The mandatory legal liability remains 
* 	unaffected. 
* ------------------------------------------------------------------------------------ 
* 	Revision History: 
* 
* 	VERSION 		DATE 			INITIALS 			DESCRIPTION 
* 	0.1 			23.05.2018 		mbo 				Created.
*	0.2				08.02.2019		mbo					Racecondition fixed +
*														Parameter Exclusion mode
* 
**************************************************************************************)
VAR_INPUT
	Execute						: BOOL; // Rising edge, starts new search process
	TU_Present					: BOOL; // TU is available
	TU_Index					: DINT; // Waiting TU data index 
	Branch						: I_BranchCheckpoint; // Branch path
	BranchExclusionMode			: BOOL := FALSE; // False = TU on a branch is possible next, TRUE = TU on a branch is excluded as possible next
	iEstimateNextService		: I_SeqEstimateNext; // Service to estimate possible next in order to save calculation time (optional)
END_VAR

VAR_OUTPUT
	Busy						: BOOL; // Process ongoing
	Error						: BOOL; // Error during process
	Release						: BOOL; // Movement released
END_VAR

VAR_IN_OUT 
	TU_Table					: ARRAY[0..Conveyor.NUMBER_OF_TU_DATA] OF ST_TU_Data; // TU Table
END_VAR

VAR
	fbTrigExecute				: R_TRIG; // Trigger new request
	State 						: INT; // State machine
	SequenceDataPresent			: BOOL; // TU consists of sequence information
	TU_IsNextInSequence			: BOOL; // Waiting TU is the next expected for that destination
	fbSeqReleaseRequest			: FB_SeqReleaseRequest; // Request release movement
	TU_DataChanged				: BOOL; // Data of blocking index has changed since it was detected, determine new
	TU_LocationChanged			: BOOL; // Location of blocking index has changed, determine new
	
	BlockingTU_Index			: DINT; // TU index of blocking index
	BlockingCheckpointID		: STRING(5); // Checkpoint ID of blocking index
	BlockingTU_ID			  	: STRING(Conveyor.TU_ID_STRINGLENGTH); // HashCode of blocking index
	BlockingAssignmentID		: UDINT; // Assignment ID of blocking index
	BlockingSequence			: ULINT; // Sequence of blocking index
	BlockingSubSequence			: DINT; // Sub sequence of blocking index
	BlockingDestination			: ST_PositionIdent; // Blocking Destination
	BlockingDestinationSlot		: INT; // Blocking Destination Slot
	BlockingHaltSequencing		: BOOL; // Halt sequence bit of blocking TU 
	SelfBlocking				: BOOL; // Tu is blocking itself
END_VAR

// Monitor new request trigger
fbTrigExecute(CLK := Execute);

CASE State OF
	// Wait for a new TU
	0:
		// Wait for new start trigger
		IF fbTrigExecute.Q THEN
			// Validate inputs
			IF Branch = 0 THEN
				Error := TRUE;
				RETURN;
			END_IF

			Busy := TRUE;
			Release := FALSE;
			TU_IsNextInSequence := FALSE;
			Error := FALSE;

			// When a requesting TU is present
			IF TU_Present THEN
				// If already a blocking TU was determined on a previous search, 
				// check if state or position has changed of it
				IF BlockingTU_Index > 0 THEN
					// Detect if the data of the monitored TU index has changed (e.g. TU data Add/Remove/Update)		
					TU_DataChanged := TU_Table[BlockingTU_Index].AssignmentID <> BlockingAssignmentID OR
									  TU_Table[BlockingTU_Index].TU_ID.ASCII <> BlockingTU_ID OR
									  TU_Table[BlockingTU_Index].DataSet.Sequence <> BlockingSequence OR
									  TU_Table[BlockingTU_Index].DataSet.SubSequence <> BlockingSubSequence OR
                                      TU_Table[BlockingTU_Index].Destination[1].eFunctionNumber <> BlockingDestination.eFunctionNumber OR
  									  TU_Table[BlockingTU_Index].Destination[1].ZoneNumber <> BlockingDestination.ZoneNumber OR
									  TU_Table[BlockingTU_Index].DataSet.DestinationSlot <> BlockingDestinationSlot OR
									  TU_Table[BlockingTU_Index].DataSet.HaltSequencing <> BlockingHaltSequencing;
			
					// Detect if the TU has changed the location (e.g. entered a new path)
					TU_LocationChanged := TU_Table[BlockingTU_Index].DataSet.CheckpointID <> BlockingCheckpointID;
					
					// If blocking index is same as requesting
					SelfBlocking := BlockingTU_Index = TU_Index;
					
					// Data changed, new release request		  
					IF TU_DataChanged OR TU_LocationChanged OR SelfBlocking THEN
						M_ClearBlockingData();
					END_IF
				END_IF

				// A TU is blocking 
				IF BlockingTU_Index > 0 THEN
					// No release, stay in state, no drive on
					Busy := FALSE;
					Release := FALSE;
					State := 0;
					
				// If the waiting TU consists of TU data,
				ELSIF TU_Index > 0 THEN
					// If the TU consists of sequencing information
					SequenceDataPresent := TU_Table[TU_Index].DataSet.Sequence > 0 AND
					                       TU_Table[TU_Index].Destination[1].eFunctionNumber > 0;
					   
					// When ever valid sequence information are avaiable, 
					// check if the TU is already available in the pre calculation service. Otherwise
					// request release.
					IF SequenceDataPresent THEN	
						// When a pre calculation service is configured and ready
						IF iEstimateNextService <> 0 THEN
							// Tu was found in precalculated list -> Release
							TU_IsNextInSequence:= iEstimateNextService.M_IsNextInSequence(
																			mTU_Index := TU_Index,
																			mTU_Data := TU_Table[TU_Index]);
																								
							IF TU_IsNextInSequence THEN
								// Release immediately, stay in state
								Busy := FALSE;
								Release := TRUE;
								State := 0;
							END_IF
						END_IF
						
						// If TU was not found in temporary next list, request release
						IF NOT TU_IsNextInSequence THEN
							// Trigger new release request
							fbSeqReleaseRequest(
								Execute:= TRUE, 
								TU_Index := TU_Index,
								Destination:= TU_Table[TU_Index].Destination[1], 
								DestinationSlot:= TU_Table[TU_Index].DataSet.DestinationSlot, 
								Sequence:= TU_Table[TU_Index].DataSet.Sequence, 
								SubSequence:= TU_Table[TU_Index].DataSet.SubSequence, 
								Branch:= Branch, 
								BranchExclusionMode := BranchExclusionMode, 
								TU_Table:= TU_Table);
		
							State := 1;	
						END_IF
					// TU without sequence information
					ELSE
						// Release immediately, stay in state
						Busy := FALSE;
						Release := TRUE;
						State := 0;
					END_IF

				// TU without data
				ELSE
					// Release immediately, stay in state
					Busy := FALSE;
					Release := TRUE;
					State := 0;
				END_IF
			// No TU Present
			ELSE
				// Release immediately, stay in state
				Busy := FALSE;
				State := 0;
			END_IF
		END_IF
	1:
		fbSeqReleaseRequest(Execute := FALSE, TU_Table:= TU_Table);
		
		// Wait until process is done to check error and result
		IF NOT fbSeqReleaseRequest.Busy THEN
			IF NOT fbSeqReleaseRequest.Error THEN
				// Release successful
				IF fbSeqReleaseRequest.Release THEN
					Busy := FALSE;
					Release := TRUE;
					
					State := 0;
				// Release not permitted, store data of next blocking TU
				ELSE
					BlockingTU_Index := fbSeqReleaseRequest.BlockingTU_Index;
					
					// When a blocking index could be determined
					IF BlockingTU_Index > 0 THEN
						BlockingAssignmentID := TU_Table[BlockingTU_Index].AssignmentID;
						BlockingTU_ID := TU_Table[BlockingTU_Index].TU_ID.ASCII;
						BlockingCheckpointID := TU_Table[BlockingTU_Index].DataSet.CheckpointID;
						BlockingSequence := TU_Table[BlockingTU_Index].DataSet.Sequence;
						BlockingSubSequence := TU_Table[BlockingTU_Index].DataSet.SubSequence;
						BlockingDestination := TU_Table[BlockingTU_Index].Destination[1];
						BlockingDestinationSlot :=  TU_Table[BlockingTU_Index].DataSet.DestinationSlot;
						BlockingHaltSequencing := TU_Table[BlockingTU_Index].DataSet.HaltSequencing;
					ELSE
						M_ClearBlockingData();
					END_IF
					
					Busy := FALSE;
					Release := FALSE;
					
					State := 0;
				END_IF
			// Error during search
			ELSE
				Error := TRUE;
				Busy  := FALSE;
				State := 0;
			END_IF
		END_IF
ELSE
	State := 0;
END_CASE

/// Clear blocking data
METHOD PROTECTED M_ClearBlockingData
VAR_INPUT
END_VAR
// Clear monitor of blocking index structure
BlockingTU_Index := 0;
BlockingAssignmentID :=0;
BlockingTU_ID := '';
BlockingCheckpointID := '';
BlockingSequence := 0;
BlockingSubSequence := 0;
BlockingDestination.eFunctionNumber := 0;
BlockingDestination.ZoneNumber := 0;
BlockingDestinationSlot :=  0;
BlockingHaltSequencing :=  FALSE;
END_METHOD

// Resets all stored information
METHOD M_Reset : BOOL
VAR_INPUT
END_VAR
M_ClearBlockingData();
END_METHOD

{attribute 'monitoring' := 'call'}
/// Recursive branch search active. Remark: No automated loop detection.
PROPERTY P_BranchRecursive : BOOL
GET
P_BranchRecursive := fbSeqReleaseRequest.P_BranchRecursive;
END_GET
SET
fbSeqReleaseRequest.P_BranchRecursive := P_BranchRecursive;
END_SET
END_PROPERTY

/// TU Entries scanned per cycle
PROPERTY P_EntriesPerCycle : DINT // Default 600
GET
P_EntriesPerCycle := fbSeqReleaseRequest.P_EntriesPerCycle;
END_GET
SET
fbSeqReleaseRequest.P_EntriesPerCycle := P_EntriesPerCycle;
END_SET
END_PROPERTY

END_FUNCTION_BLOCK

// ---- 20_Product/30_Toolbox/16_Sequencing/10_Core/FB_SeqReleaseRequest.TcPOU
/// Validates a request of a TU to get permission to release movement. If its not 
/// possible, the TU index of the blocking TU is returned.
///
/// Blocking TU = A TU with a lower Sequence/Subsequence pair
///	              which is not located in system or is found on branch.
/// Requires multiple cycles, check busy signal
FUNCTION_BLOCK FB_SeqReleaseRequest
(************************************************************************************** 
* 	Application 		: BoxControl Framework 
* 	Revision 			: $Revision: 404877 $ 
* 	Revision date 		: $Date: 2018-04-26 14:10:34 +0200 (Thu, 26 Apr 2018) $ 
* 	Last changed by 	: $Author: b7ernsb $ 
* 	URL 				: $URL: http://almscdc.swisslog.com/repo/SWPD/Development/BoxControlFramework/21_Projects/BCF_2.0/trunk/BCF/BCF/JumpStart/20_Product/10_App/12_E_Functions/10_Lib/10_Conv/FB_FunctionConv.TcPOU $ 
* ------------------------------------------------------------------------------------ 
* 	© Swisslog AG 
* 	Swisslog is not liable for any usage of this source code that is not agreed 
* 	on between Swisslog and the other party. The mandatory legal liability remains 
* 	unaffected. 
* ------------------------------------------------------------------------------------ 
* 	Revision History: 
* 
* 	VERSION 		DATE 			INITIALS 			DESCRIPTION 
* 	0.1 			01.05.2018 		mbo 				Created.
*	0.2				08.02.2019		mbo					Checkpoint of blocking added
*														+ Branch exclusion mode
* 
**************************************************************************************)
VAR_INPUT
	Execute						: BOOL; // Rising edge, starts new search process
	TU_Index					: DINT; // Requesting TU Index
	Destination					: ST_PositionIdent; // Destination of requesting Sequence
	DestinationSlot				: INT; // Destination slot of requesting Sequence
	Sequence					: ULINT; // Requesting sequence
	SubSequence					: DINT; // Requesting sub sequence
	Branch						: I_BranchCheckpoint; // Branch to check
	BranchExclusionMode			: BOOL := FALSE; // False = TU on a branch is possible next, TRUE = TU on a branch is excluded as possible next
END_VAR
VAR_OUTPUT
	Busy						: BOOL; // Process ongoing
	Release 					: BOOL; // Allowed to release
	BlockingTU_Index			: DINT; // Blocking TU-Index for the requesting sequence
	BlockingTU_Checkpoint		: STRING(5); // Data of blocking TU
	Error 						: BOOL; // Error (Configuration or invalid result), Reset with new trigger
END_VAR
VAR_IN_OUT
	TU_Table					: ARRAY[0..Conveyor.NUMBER_OF_TU_DATA] OF ST_TU_Data; // TU Table
END_VAR
VAR
	EntriesPerCycle				: DINT := SequencingParameter.SCAN_ENTRIES_PER_CYCLE; // Entries scanned per cylce
	EntryIdx					: DINT; // Entry iterator
	MinArrayIndex				: DINT; // Minimum index of TU Array
	MaxArrayIndex				: DINT; // Maximum index of TU Array
	StartIndex					: DINT; // Start index of current iteration
	EndIndex					: DINT; // End index of current iteration
	IterationCounter			: DINT; // Iteration counter
	
	CurrentBlockingTU_Index		: DINT; // Current blocking TU index
	State						: INT; // State machine, 0=Idle, 1 = Search
	fbTrigExecute				: R_TRIG; // Trigger new request
	BranchRecursive				: BOOL := TRUE; // Recursive branch search active (Default = True)
	FoundOnBranch				: BOOL; // Checkpoint ID found on one of the configured branches
	LowestBlockingSequence		: ULINT; // Lowest blocking sequence number
	LowestBlockingSubSequence	: DINT; // Lowest blocking sub sequence number
	rTU_DataEntry				: REFERENCE TO ST_TU_Data; // Currently checked entry
END_VAR

// Monitor new request trigger
fbTrigExecute(CLK := Execute);

CASE State OF
	// Idle - State
	0:
		// Wait for new start trigger
		IF fbTrigExecute.Q THEN
			// Check inputs
			IF Sequence = 0 OR
			  TU_Index = 0 OR
			   Destination.eFunctionNumber = E_FunctionNumber.F_BEGIN_FUNCTION OR
			   Branch = 0 THEN
			   // Invalid inputs
			   Error := TRUE;
			   RETURN;
			END_IF
			
			// Initialize 
			Error := FALSE;
			Busy := TRUE;
			Release := FALSE;
			IterationCounter := 0;
			BlockingTU_Index := 0;
			BlockingTU_Checkpoint := '';
			CurrentBlockingTU_Index := 0;
			
			// Only search when sequencing is not on hold for this TU 	
			IF NOT TU_Table[TU_Index].DataSet.HaltSequencing THEN
				// Set lowest values to actual
				LowestBlockingSequence := Sequence;
				LowestBlockingSubSequence := SubSequence;
				
				MinArrayIndex := 1; //LOWER_BOUND(TU_Table,1);
				MaxArrayIndex := Conveyor.NUMBER_OF_TU_DATA; //UPPER_BOUND(TU_Table,1);
				
				State := 1;
			ELSE 
				Busy := FALSE;			
				State := 0;
			END_IF
		END_IF
		
	// Iterate over multiple cycles through TU Table	
	1:
		StartIndex := MinArrayIndex + IterationCounter * EntriesPerCycle;
		EndIndex   := StartIndex + EntriesPerCycle;
	
		FOR EntryIdx := StartIndex TO EndIndex DO
			
			// Scan of TU Table completed
			IF EntryIdx > MaxArrayIndex THEN
				// If no blocking index was found, release immediatley
				IF CurrentBlockingTU_Index = 0 THEN	
					BlockingTU_Index := 0;
					BlockingTU_Checkpoint := '';
					
					Release := TRUE;
					
				// Otherwise, ensure found index is still valid
				ELSE
					IF M_IsFoundBlockingIndexValid(TU_Table) THEN
						BlockingTU_Index := CurrentBlockingTU_Index;
						BlockingTU_Checkpoint := TU_Table[BlockingTU_Index].DataSet.CheckpointID;
						
						Release := FALSE;
					ELSE
						BlockingTU_Index := 0;
						BlockingTU_Checkpoint := '';
						
						// Result not valid, new search required
						Error := TRUE;
						Release := FALSE;
					END_IF
				END_IF
				
				Busy := FALSE;
				
				State := 0;
				RETURN;
			END_IF
			
			rTU_DataEntry REF= TU_Table[EntryIdx];
			
			// Skip this loop if...
            // - own index is found
            // - Empty data set is found
			// - Data set without job present is found ( no destination)
			IF EntryIdx = TU_Index OR 
               NOT rTU_DataEntry.DataSet.DataPresent OR 
               NOT rTU_DataEntry.DataSet.JobPresent THEN
				CONTINUE;
			END_IF

			// Check if TU has same Destination and Destination slot, 
			// otherwise it is not relevant for sequence of requesting TU
			IF rTU_DataEntry.Destination[1].eFunctionNumber = Destination.eFunctionNumber AND
			   rTU_DataEntry.Destination[1].ZoneNumber = Destination.ZoneNumber THEN
				IF rTU_DataEntry.DataSet.DestinationSlot = DestinationSlot THEN
					
					// TU's with a higher sequence number than the requesting or 0 are not
					// taked into account of sequencing -> Skip
					
					// TU's can be ignored if...
					// - Sequence is 0 and is therefore not part of a sequence
					// - Sequence is equal to requesting, but subsequence is higher
					// - Sequence is higher than an already found lower sequence
					
					IF  rTU_DataEntry.DataSet.Sequence = 0 OR
					   (rTU_DataEntry.DataSet.Sequence = LowestBlockingSequence AND
					    rTU_DataEntry.DataSet.SubSequence > LowestBlockingSubSequence) OR
					   (rTU_DataEntry.DataSet.Sequence > LowestBlockingSequence) THEN

						// Skip
						;
				
					// TU is in range for a possible blocking TU
					ELSE
						// When the currently checked TU has the same sequence number
						// as the last found blocking sequence number, only sub sequence 
						// needs to be checked further
						IF rTU_DataEntry.DataSet.Sequence = LowestBlockingSequence THEN
							// Only lower sub sequences are checked for blocking
							IF rTU_DataEntry.DataSet.SubSequence < LowestBlockingSubSequence THEN
								// Check if current comapared TU is blocking
								IF 	M_IsTU_Blocking(rTU_DataEntry) THEN
									LowestBlockingSubSequence := rTU_DataEntry.DataSet.SubSequence;
								   	// Store blocking index
							   		CurrentBlockingTU_Index := EntryIdx;
									
								// Otherwise the found TU is not influence sequencing of requesting
								ELSE
								   // Skip
								   ;
								END_IF
							END_IF
					
						// Sequence number is lower than last found blocking sequence
						ELSE
							// Check if current comapared TU is blocking
							IF 	M_IsTU_Blocking(rTU_DataEntry) THEN
							   // TU is blocking, update Lowest blocking sequence pair
							   LowestBlockingSequence := rTU_DataEntry.DataSet.Sequence;
							   LowestBlockingSubSequence := rTU_DataEntry.DataSet.SubSequence;
							   
							   // Store blocking index
							   CurrentBlockingTU_Index := EntryIdx;
							END_IF
						END_IF
					END_IF
				END_IF
			END_IF
		END_FOR

		IterationCounter := IterationCounter + 1;
ELSE
	// Default
	State := 0;
END_CASE

/// Check if current comapared TU is:
/// - Not located,
/// - Found on branch (Default mode) or Not found on a branch (Exclusion mode) 
/// Sequencing is temporarily haltet for this TU				
/// so its a possible next TU
METHOD PROTECTED M_IsTU_Blocking : BOOL // Returns true if blocking
VAR_INPUT
	mrTU_DataEntry		: REFERENCE TO ST_TU_Data; // Currently checked entry
END_VAR
VAR
	mFoundOnBranch		: BOOL;
END_VAR
M_IsTU_Blocking := FALSE;

// Ensure it is still a problem for the branch	
mFoundOnBranch := Branch.M_IsOnBranches(BranchRecursive, mrTU_DataEntry.DataSet.CheckpointID);

IF (mFoundOnBranch AND NOT BranchExclusionMode) OR
   (NOT mFoundOnBranch AND BranchExclusionMode) OR
   (mrTU_DataEntry.DataSet.CheckpointID = '') OR
    mrTU_DataEntry.DataSet.HaltSequencing THEN
   
   M_IsTU_Blocking := TRUE;
END_IF
END_METHOD

/// This method checks if found index is still valid after a search over multiple cycles, 
/// because during search the state of index could have changed (Race condition).
METHOD PROTECTED M_IsFoundBlockingIndexValid : BOOL // Returns true if still valid, otherwise false
VAR_IN_OUT
	mTU_Table				: ARRAY[0..Conveyor.NUMBER_OF_TU_DATA] OF ST_TU_Data;
END_VAR
VAR
	mrTU_DataEntry			: REFERENCE TO ST_TU_Data; // Currently checked entry
END_VAR
VAR_INST
	SequenceDataPresent		: BOOL; // Sequence data present
	TU_IsPartOfDestSequence	: BOOL; // Sequence data are for requested destination
END_VAR
M_IsFoundBlockingIndexValid := FALSE;

// Validate inputs
IF CurrentBlockingTU_Index <= 0 THEN
	RETURN;
END_IF

mrTU_DataEntry REF= mTU_Table[CurrentBlockingTU_Index];

// Check reference is valid
IF NOT __ISVALIDREF(mrTU_DataEntry) THEN
	RETURN;
END_IF

// Validate its TU data
// - Sequencing, 
// - Part of that sequence (destination)
// - Still at the detected checkpoint
SequenceDataPresent := mrTU_DataEntry.DataSet.Sequence > 0 AND
					   mrTU_DataEntry.Destination[1].eFunctionNumber > 0;
					   
TU_IsPartOfDestSequence := mrTU_DataEntry.Destination[1].eFunctionNumber = Destination.eFunctionNumber AND
						   mrTU_DataEntry.Destination[1].ZoneNumber = Destination.ZoneNumber AND
						   mrTU_DataEntry.DataSet.DestinationSlot = DestinationSlot;

IF SequenceDataPresent AND
   TU_IsPartOfDestSequence THEN	

	M_IsFoundBlockingIndexValid := M_IsTU_Blocking(rTU_DataEntry);
END_IF
END_METHOD

{attribute 'monitoring' := 'call'}
/// Recursive branch search active. Remark: No automated loop detection.
PROPERTY P_BranchRecursive : BOOL
GET
P_BranchRecursive := BranchRecursive;
END_GET
SET
BranchRecursive := P_BranchRecursive;
END_SET
END_PROPERTY

/// TU Entries scanned per cycle
PROPERTY P_EntriesPerCycle : DINT // Default 600
SET
EntriesPerCycle := P_EntriesPerCycle;
END_SET
GET
P_EntriesPerCycle := EntriesPerCycle;
END_GET
END_PROPERTY

END_FUNCTION_BLOCK

// ---- 20_Product/30_Toolbox/16_Sequencing/10_Core/FB_SeqBranchMux.TcPOU
/// Branch multiplexer. Allows to multiplex several branches.
/// This is no checkpoint! Automated update of checkpoint id is not possible, needs to be done manually.
/// Remark: No automated loop detection
FUNCTION_BLOCK FB_SeqBranchMux IMPLEMENTS I_BranchCheckpoint
(************************************************************************************** 
* 	Application 		: BoxControl Framework 
* 	Revision 			: $Revision: 404877 $ 
* 	Revision date 		: $Date: 2018-04-26 14:10:34 +0200 (Thu, 26 Apr 2018) $ 
* 	Last changed by 	: $Author: b7ernsb $ 
* 	URL 				: $URL: http://almscdc.swisslog.com/repo/SWPD/Development/BoxControlFramework/21_Projects/BCF_2.0/trunk/BCF/BCF/JumpStart/20_Product/10_App/12_E_Functions/10_Lib/10_Conv/FB_FunctionConv.TcPOU $ 
* ------------------------------------------------------------------------------------ 
* 	© Swisslog AG 
* 	Swisslog is not liable for any usage of this source code that is not agreed 
* 	on between Swisslog and the other party. The mandatory legal liability remains 
* 	unaffected. 
* ------------------------------------------------------------------------------------ 
* 	Revision History: 
* 
* 	VERSION 		DATE 			INITIALS 			DESCRIPTION 
* 	0.1 			23.05.2018 		mbo 				Created.
* 
**************************************************************************************)
VAR_INPUT
	BranchRecursive 	: BOOL := FALSE; // Check all connected recursive (Default = FALSE)
	BranchA				: I_BranchCheckpoint; // Branch to check
	BranchB				: I_BranchCheckpoint; // Branch to check
	BranchC				: I_BranchCheckpoint; // Branch to check
	BranchD				: I_BranchCheckpoint; // Branch to check
END_VAR
VAR
	Empty				: STRING(5) := ''; // Empty string to fullfil interface
END_VAR

;

/// Searches if a checkpoint can be found on a specific branch
/// Returns true if found, false = not found 
METHOD M_IsOnBranches : BOOL
VAR_INPUT
	mRecursive	: BOOL := FALSE;// Search recursive through the whole tree
END_VAR
VAR_IN_OUT CONSTANT
	mCheckpointID	: STRING(5); // Last checkpoint id	
END_VAR

IF BranchA <> 0 THEN
	 IF BranchA.M_IsOnBranches(BranchRecursive, mCheckpointId) THEN;
	 	M_IsOnBranches := TRUE;
		RETURN;
	END_IF
END_IF

IF BranchB <> 0 THEN
	 IF BranchB.M_IsOnBranches(BranchRecursive, mCheckpointId) THEN;
	 	M_IsOnBranches := TRUE;
		RETURN;
	END_IF
END_IF

IF BranchC <> 0 THEN
	 IF BranchC.M_IsOnBranches(BranchRecursive, mCheckpointId) THEN;
	 	M_IsOnBranches := TRUE;
		RETURN;
	END_IF
END_IF

IF BranchD <> 0 THEN
	 IF BranchD.M_IsOnBranches(BranchRecursive, mCheckpointId) THEN;
	 	M_IsOnBranches := TRUE;
		RETURN;
	END_IF
END_IF
END_METHOD

/// Identifier for checkpoint
{attribute 'monitoring' := 'call'}
{attribute 'suppress_wrn_C0410'}
PROPERTY P_CheckpointID : REFERENCE TO STRING(5)
GET
P_CheckpointID REF= Empty;
END_GET
END_PROPERTY

END_FUNCTION_BLOCK

// ---- 20_Product/30_Toolbox/16_Sequencing/10_Core/FB_SeqBuildStream.TcPOU
/// Builds a list of TUs of one stream considering configured branch
/// Remark: Request sequence information are included.
FUNCTION_BLOCK FB_SeqBuildStream
(************************************************************************************** 
* 	Application 		: BoxControl Framework 
* 	Revision 			: $Revision: 404877 $ 
* 	Revision date 		: $Date: 2018-04-26 14:10:34 +0200 (Thu, 26 Apr 2018) $ 
* 	Last changed by 	: $Author: b7ernsb $ 
* 	URL 				: $URL: http://almscdc.swisslog.com/repo/SWPD/Development/BoxControlFramework/21_Projects/BCF_2.0/trunk/BCF/BCF/JumpStart/20_Product/10_App/12_E_Functions/10_Lib/10_Conv/FB_FunctionConv.TcPOU $ 
* ------------------------------------------------------------------------------------ 
* 	© Swisslog AG 
* 	Swisslog is not liable for any usage of this source code that is not agreed 
* 	on between Swisslog and the other party. The mandatory legal liability remains 
* 	unaffected. 
* ------------------------------------------------------------------------------------ 
* 	Revision History: 
* 
 * VERSION DATE         INITIALS     DESCRIPTION
 * 0.0     DD.MM.YYYY   (name)       (explain customized modifications)
* 
**************************************************************************************)
VAR_INPUT
	Execute						: BOOL; // Rising edge, starts new search process
	Destination					: ST_PositionIdent; // Destination of stream to build
	DestinationSlot				: INT; // Destination slot of stream to build
	BranchExclusionMode			: BOOL := FALSE; // False = TU on a branch is possible next, TRUE = TU on a branch is excluded as possible next
	Branch						: I_BranchCheckpoint; // Branch to check
END_VAR
VAR_OUTPUT
	Busy						: BOOL; // Process ongoing
	EntryCounter				: INT; // Entries in range list
	NextTU_Index				: DINT; // Next expected TU_Index which is not located or found on branch (First of list)
	NextTU_Checkpoint			: STRING(5); // Checkpoint location of next TU at point when it was detected
	StreamList					: ARRAY[1..MAX_Stream_LIST] OF ST_SeqEntry; // Stream list of TUs, priority ascending (1 = First)
	Error 						: BOOL; // Error configuration, Reset with new trigger
END_VAR
VAR_IN_OUT
	TU_Table					: ARRAY[0..Conveyor.NUMBER_OF_TU_DATA] OF ST_TU_Data; // TU Table
END_VAR
VAR
	EntriesPerCycle				: DINT := SequencingParameter.SCAN_ENTRIES_PER_CYCLE; // Entries scanned per cylce
	EntryIdx					: DINT; // Entry iterator
	MinArrayIndex				: DINT; // Minimum index of TU Array
	MaxArrayIndex				: DINT; // Maximum index of TU Array
	StartIndex					: DINT; // Start index of current iteration
	EndIndex					: DINT; // End index of current iteration
	IterationCounter			: DINT; // Iteration counter
	FoundOnBranch				: BOOL; // Checkpoint ID found on one of the configured branches
	BranchRecursive				: BOOL := TRUE; // Recursive branch search active (Default = True)
	State						: INT; // State machine, 0=Idle, 1 = Search
	fbTrigExecute				: R_TRIG; // Trigger new request
	rTU_DataEntry				: REFERENCE TO ST_TU_Data; // Currently checked entry
END_VAR
VAR CONSTANT
	MAX_STREAM_LIST				: INT := SequencingParameter.MAX_STREAMBUILDER_LIST; // Max limit of entries
END_VAR

// Monitor new request trigger
fbTrigExecute(CLK := Execute);

CASE State OF
	// Idle - State
	0:
		// Wait for new start trigger
		IF fbTrigExecute.Q THEN
			// Validate inputs
			IF Destination.eFunctionNumber = E_FunctionNumber.F_BEGIN_FUNCTION OR
			   Branch = 0 THEN
			   // Invalid inputs
			   Error := TRUE;
			   RETURN;
			END_IF
			
			// Initialize 
			Error := FALSE;
			Busy := TRUE;
			
			// Clear range list
			MEMSET(ADR(StreamList), 0, SIZEOF(StreamList));

			IterationCounter := 0;
			NextTU_Index := 0;
			NextTU_Checkpoint := '';
			
			MinArrayIndex := 1; //LOWER_BOUND(TU_Table,1);
			MaxArrayIndex := Conveyor.NUMBER_OF_TU_DATA; //UPPER_BOUND(TU_Table,1);
			State := 1;
		END_IF
		
	// Iterate over multiple cycles through TU Table	
	1:
		StartIndex := MinArrayIndex + IterationCounter * EntriesPerCycle;
		EndIndex   := StartIndex + EntriesPerCycle;
	
		FOR EntryIdx := StartIndex TO EndIndex DO
			// When scan is completed
			IF EntryIdx > MaxArrayIndex THEN
				
				IF StreamList[1].TU_Index = 0 THEN
					NextTU_Checkpoint := '';
					NextTU_Index := 0;
				// Otherwise, validate found indexes
				ELSE
					// Get index and checkpoint of next tu
					NextTU_Index := M_GetValidNextIndex(TU_Table);
					
					IF NextTU_Index > 0 THEN
						NextTU_Checkpoint := TU_Table[NextTU_Index].DataSet.CheckpointID;
					ELSE
						NextTU_Checkpoint := '';
					END_IF
				END_IF
				
				Busy := FALSE;
			
				State := 0;
				RETURN;
			END_IF
			
			rTU_DataEntry REF= TU_Table[EntryIdx];
			
			// Skip this loop if...
            // - Empty data set is found
			// - Data set without job present is found ( no destination)
            IF NOT rTU_DataEntry.DataSet.DataPresent OR 
               NOT rTU_DataEntry.DataSet.JobPresent THEN
				CONTINUE;
			END_IF
			
			// Check if TU has same Destination and Destination slot, 
			// otherwise it is not relevant for sequencing of requesting TU
			IF rTU_DataEntry.Destination[1].eFunctionNumber = Destination.eFunctionNumber AND
			   rTU_DataEntry.Destination[1].ZoneNumber = Destination.ZoneNumber THEN
				IF rTU_DataEntry.DataSet.DestinationSlot = DestinationSlot THEN
					
					// TU's can be ignored if...
					// - Sequence is 0 and is therefore not part of a sequence
					IF rTU_DataEntry.DataSet.Sequence = 0 THEN
						// Skip
						;
				
					// Sequence is in a valid range for a possible next
					// - All TU's with same destination AND
					// - Higher sequence information than requesting
					// - AND (NOT)* on Branch  
					//   * based on mode (Default, Exclusion)
					ELSE
						// Check if current comapared TU is:
						// - Not located,
						// - Found on branch (Default mode) or Not found on a branch (Exclusion mode) 
						// Sequencing is temporarily haltet for this TU
						// so its a possible next TU
						FoundOnBranch := Branch.M_IsOnBranches(BranchRecursive, rTU_DataEntry.DataSet.CheckpointId);
						
						IF 	(FoundOnBranch AND NOT BranchExclusionMode) OR
							(NOT FoundOnBranch AND BranchExclusionMode) OR
						  	rTU_DataEntry.DataSet.CheckpointID = '' OR
							rTU_DataEntry.DataSet.HaltSequencing THEN
						   // TU is possible next, update range list
						   M_AddToStreamList(EntryIdx, rTU_DataEntry);
						END_IF
					END_IF
				END_IF
			END_IF
		END_FOR

		IterationCounter := IterationCounter + 1;
ELSE
	// Default
	State := 0;
END_CASE

/// Add Entry sorted to Range list.
METHOD PRIVATE M_AddToStreamList
VAR_INPUT
	mTU_Index	: DINT; // TU index which should be added
END_VAR
VAR_IN_OUT
	mTU_Data	: ST_TU_Data; // TU data set to add
END_VAR
VAR
	mIdx		: INT; // Iterator
END_VAR

FOR mIdx := 1 TO MAX_STREAM_LIST DO
	// If slot is empty, take over data
	IF StreamList[mIdx].TU_Index = 0 THEN
		StreamList[mIdx].TU_Index := mTU_Index;
		StreamList[mIdx].Sequence := mTU_Data.DataSet.Sequence;
		StreamList[mIdx].SubSequence := mTU_Data.DataSet.SubSequence;
		StreamList[mIdx].Destination := mTU_Data.Destination[1];
		StreamList[mIdx].DestinationSlot := mTU_Data.DataSet.DestinationSlot;
		StreamList[mIdx].TU_ID_HashCode := mTU_Data.TU_ID.HashCode;
		StreamList[mIdx].TU_ID := mTU_Data.TU_ID.ASCII;
		StreamList[mIdx].AssignmentID := mTU_Data.AssignmentID;
		StreamList[mIdx].CheckpointID := mTU_Data.DataSet.CheckpointID;
	
		EntryCounter := EntryCounter + 1;
		EXIT;
	ELSE
		// When requesting Sequence information are equal, compare subsequence
		IF mTU_Data.DataSet.Sequence = StreamList[mIdx].Sequence THEN
			// If sub sequence is lower, replace and shift list
			IF mTU_Data.DataSet.SubSequence < StreamList[mIdx].SubSequence THEN
				//Shift list
				M_ShiftAndClearSlot(mIdx);
				// Insert new data set, with all relevant data, to validate later
				StreamList[mIdx].TU_Index := mTU_Index;
				StreamList[mIdx].Sequence := mTU_Data.DataSet.Sequence;
				StreamList[mIdx].SubSequence := mTU_Data.DataSet.SubSequence;
				StreamList[mIdx].Destination := mTU_Data.Destination[1];
				StreamList[mIdx].DestinationSlot := mTU_Data.DataSet.DestinationSlot;
				StreamList[mIdx].TU_ID_HashCode := mTU_Data.TU_ID.HashCode;
				StreamList[mIdx].TU_ID := mTU_Data.TU_ID.ASCII;
				StreamList[mIdx].AssignmentID := mTU_Data.AssignmentID;
				StreamList[mIdx].CheckpointID := mTU_Data.DataSet.CheckpointID;
				
				EntryCounter := EntryCounter + 1;
				EXIT;
			END_IF	
		// When requesting Sequence information are lower or equal
		ELSIF mTU_Data.DataSet.Sequence <= StreamList[mIdx].Sequence THEN
			//Shift list
			M_ShiftAndClearSlot(mIdx);
			// Insert new data set, with all relevant data, to validate later
			StreamList[mIdx].TU_Index := mTU_Index;
			StreamList[mIdx].Sequence := mTU_Data.DataSet.Sequence;
			StreamList[mIdx].SubSequence := mTU_Data.DataSet.SubSequence;
			StreamList[mIdx].Destination := mTU_Data.Destination[1];
			StreamList[mIdx].DestinationSlot := mTU_Data.DataSet.DestinationSlot;
			StreamList[mIdx].TU_ID_HashCode := mTU_Data.TU_ID.HashCode;
			StreamList[mIdx].TU_ID := mTU_Data.TU_ID.ASCII;
			StreamList[mIdx].AssignmentID := mTU_Data.AssignmentID;
			StreamList[mIdx].CheckpointID := mTU_Data.DataSet.CheckpointID;
			
			EntryCounter := EntryCounter + 1;
			EXIT;	
		END_IF
	END_IF
END_FOR
END_METHOD

// Returns next valid tu index
// Remark: This check is required after the search over multiple cycles, 
// because during search the state of index could have changed (Race condition).
METHOD PROTECTED M_GetValidNextIndex : DINT // 0= No next index, >0 Next TU Index
VAR_IN_OUT
	mTU_Table					: ARRAY[0..Conveyor.NUMBER_OF_TU_DATA] OF ST_TU_Data; // TU Table
END_VAR
VAR
	mIdx					: INT; // Iterator
	mrTU_DataEntry			: REFERENCE TO ST_TU_Data; // Currently checked entry
END_VAR
VAR_INST
	NextIndex				: DINT; // Nextindex to be checked
	SequenceDataPresent		: BOOL; // Sequence data present
	TU_IsPartOfDestSequence	: BOOL; // Sequence data are for requested destination
END_VAR
M_GetValidNextIndex := 0;

IF EntryCounter = 0 THEN
	RETURN;
END_IF

// Get highest prioritized next tu index
FOR mIdx := 1 TO EntryCounter DO
	
	NextIndex := StreamList[mIdx].TU_Index;
	
	IF NextIndex = 0 THEN
		RETURN;
	END_IF
	
	mrTU_DataEntry REF= mTU_Table[NextIndex];
	
	// Check reference is valid
	IF NOT __ISVALIDREF(mrTU_DataEntry) THEN
		RETURN;
	END_IF
	
	// Validate its TU data
	// - Sequencing, 
	// - Part of that sequence (destination)
	// - Still at the detected checkpoint
	SequenceDataPresent := mrTU_DataEntry.DataSet.Sequence > 0 AND
						   mrTU_DataEntry.Destination[1].eFunctionNumber > 0;
						   
	TU_IsPartOfDestSequence := mrTU_DataEntry.Destination[1].eFunctionNumber = Destination.eFunctionNumber AND
							   mrTU_DataEntry.Destination[1].ZoneNumber = Destination.ZoneNumber AND
							   mrTU_DataEntry.DataSet.DestinationSlot = DestinationSlot;
	
	IF SequenceDataPresent AND
       TU_IsPartOfDestSequence THEN			   
		IF M_IsTU_Next(mrTU_DataEntry) THEN
		   M_GetValidNextIndex := NextIndex;
		   EXIT;
		END_IF
	END_IF
END_FOR
END_METHOD

/// Check if current comapared TU is:
/// - Not located,
/// - Found on branch (Default mode) or Not found on a branch (Exclusion mode) 
/// Sequencing is temporarily haltet for this TU				
/// so its a possible next TU
METHOD PROTECTED M_IsTU_Next : BOOL // Returns true if it is a possible next
VAR_INPUT
	mrTU_DataEntry		: REFERENCE TO ST_TU_Data; // Currently checked entry
END_VAR
VAR
	mFoundOnBranch		: BOOL;
END_VAR
M_IsTU_Next := FALSE;

// Ensure it is still a problem for the branch	
mFoundOnBranch := Branch.M_IsOnBranches(BranchRecursive, mrTU_DataEntry.DataSet.CheckpointID);

IF (mFoundOnBranch AND NOT BranchExclusionMode) OR
   (NOT mFoundOnBranch AND BranchExclusionMode) OR
   (mrTU_DataEntry.DataSet.CheckpointID = '') OR
    mrTU_DataEntry.DataSet.HaltSequencing THEN
   
   M_IsTU_Next := TRUE;
END_IF
END_METHOD

/// Checks whether a TU is part of stream list or not. 
METHOD M_IsTU_OnStream : BOOL // Returns True if found in stream list
VAR_INPUT
	mRangeLimit		: INT; // Specifies how many entries of the list serve as valid. (0=All available)
	mTU_Index		: DINT; // Requesting TU Index
END_VAR
VAR_IN_OUT
	mTU_Data			: ST_TU_Data; // Tu Data
END_VAR
VAR
	mIdx				: INT; // Iterator
	mMax				: INT; // Max entries
END_VAR
M_IsTU_OnStream := FALSE;

// Check inputs
IF mTU_Index = 0 THEN
	RETURN;
END_IF

IF mRangeLimit > 0 THEN
	mMax := mRangeLimit;
ELSE
	mMax := EntryCounter;
END_IF

// Check border
IF mMax > MAX_STREAM_LIST THEN
	mMax := MAX_STREAM_LIST;
ELSIF mMax < 1 THEN
	mMax := 1;
END_IF

FOR mIdx := 1 TO mMax DO
	// Check if an index is recorded as next
	IF mTU_Index = StreamList[mIdx].TU_Index THEN
		/// Ensure that recorded tu data entry is still the same as requesting Tu data
		IF mTU_Data.DataSet.Sequence = StreamList[mIdx].Sequence AND
		   mTU_Data.DataSet.SubSequence = StreamList[mIdx].SubSequence AND
		   mTU_Data.TU_ID.ASCII = StreamList[mIdx].TU_ID AND
		   mTU_Data.Destination[1].eFunctionNumber = StreamList[mIdx].Destination.eFunctionNumber AND
		   mTU_Data.Destination[1].ZoneNumber = StreamList[mIdx].Destination.ZoneNumber AND 
		   mTU_Data.DataSet.DestinationSlot = StreamList[mIdx].DestinationSlot THEN
		   
			M_IsTU_OnStream := TRUE;
			RETURN;
		END_IF	
	END_IF
END_FOR
END_METHOD

/// Shift entries and update entry counter
METHOD PRIVATE M_ShiftAndClearSlot : BOOL
VAR_INPUT
	mListIdx		: INT; // Index to be moved
END_VAR
VAR_INST
	NoError					: BOOL; // No error during process
	LastSlotInUse			: BOOL; // Last slot was already in use
	SizeOneSlot				: UDINT; // Size in bytes of one slot
	NumberOfBytes			: UDINT; // Number of bytes
	NumberOfEntriesToShift	: INT; // Number of entries to shift
END_VAR
// Init values
LastSlotInUse := FALSE;

// Shift following entries
IF mListIdx <= EntryCounter THEN
   
	SizeOneSlot	:= SIZEOF(StreamList[1]);

	// Check if last slot is already in use
	IF StreamList[MAX_STREAM_LIST].TU_Index <> 0 THEN
		LastSlotInUse := TRUE;
	END_IF
	
	// Calculate entries which need to be shifted
	NumberOfEntriesToShift := EntryCounter - mListIdx + 1;
	
	// Check based on the destination, if the amount of entries would exceed memory area
	IF mListIdx + NumberOfEntriesToShift > MAX_STREAM_LIST THEN
		NumberOfEntriesToShift := MAX_STREAM_LIST - mListIdx;
	END_IF 
	
	IF NumberOfEntriesToShift > 0 THEN
		NumberOfBytes :=  INT_TO_UDINT(NumberOfEntriesToShift)* SizeOneSlot;
		NoError := MEMCPY(ADR(StreamList[mListIdx+1]), ADR(StreamList[mListIdx]), NumberOfBytes) > 0;
	END_IF
	
	// Clear entry afterwards
	NoError := MEMSET(ADR(StreamList[mListIdx]), 0, SizeOneSlot) > 0 AND NoError;
	
	// If last slot was moved out of the list, decrease entry counter
	IF NoError AND LastSlotInUse THEN
		EntryCounter := EntryCounter - 1;
		
		IF EntryCounter < 0 THEN
			EntryCounter := 0;
		END_IF
	END_IF
	
	M_ShiftAndClearSlot := NoError;
ELSE
	M_ShiftAndClearSlot := TRUE;
END_IF
END_METHOD

{attribute 'monitoring' := 'call'}
/// Recursive branch search active. Remark: No automated loop detection.
PROPERTY P_BranchRecursive : BOOL
GET
P_BranchRecursive := BranchRecursive;
END_GET
SET
BranchRecursive := P_BranchRecursive;
END_SET
END_PROPERTY

END_FUNCTION_BLOCK

// ---- 20_Product/30_Toolbox/16_Sequencing/10_Core/FB_SeqGetNextTU.TcPOU
/// Returns next TU which is expected after the requesting sequence information.
/// Valid next TU : TU location unknow, or found (Default) /not found (Exception mode) on a branch
FUNCTION_BLOCK FB_SeqGetNextTU
(************************************************************************************** 
* 	Application 		: BoxControl Framework 
* 	Revision 			: $Revision: 404877 $ 
* 	Revision date 		: $Date: 2018-04-26 14:10:34 +0200 (Thu, 26 Apr 2018) $ 
* 	Last changed by 	: $Author: b7ernsb $ 
* 	URL 				: $URL: http://almscdc.swisslog.com/repo/SWPD/Development/BoxControlFramework/21_Projects/BCF_2.0/trunk/BCF/BCF/JumpStart/20_Product/10_App/12_E_Functions/10_Lib/10_Conv/FB_FunctionConv.TcPOU $ 
* ------------------------------------------------------------------------------------ 
* 	© Swisslog AG 
* 	Swisslog is not liable for any usage of this source code that is not agreed 
* 	on between Swisslog and the other party. The mandatory legal liability remains 
* 	unaffected. 
* ------------------------------------------------------------------------------------ 
* 	Revision History: 
* 
* 	VERSION 		DATE 			INITIALS 			DESCRIPTION 
* 	0.1 			03.05.2018 		mbo 				Created.
*	0.2				08.02.2019		mbo 				Checkpoint of next included
* 
**************************************************************************************)
VAR_INPUT
	Execute						: BOOL; // Rising edge, starts new search process
	TU_Index					: DINT; // Requesting TU Index
	Destination					: ST_PositionIdent; // Destination of requesting Sequence
	DestinationSlot				: INT; // Destination slot of requesting Sequence
	Sequence					: ULINT; // Requesting sequence
	SubSequence					: DINT; // Requesting sub sequence
	BranchExclusionMode			: BOOL := FALSE; // False = TU on a branch is possible next, TRUE = TU on a branch is excluded as possible next
	Branch						: I_BranchCheckpoint; // Branch to check
END_VAR
VAR_OUTPUT
	Busy						: BOOL; // Process ongoing
	NextTU_Index				: DINT; // Next expected TU_Index which is not located or found on branch
	NextTU_Checkpoint			: STRING(5); // Checkpoint location of next TU at point when it was detected
	Error 						: BOOL; // Error configuration or invalid result, Reset with new trigger
END_VAR
VAR_IN_OUT
	TU_Table					: ARRAY[0..Conveyor.NUMBER_OF_TU_DATA] OF ST_TU_Data; // TU Table
END_VAR
VAR
	EntriesPerCycle				: DINT := SequencingParameter.SCAN_ENTRIES_PER_CYCLE; // Entries scanned per cylce
	EntryIdx					: DINT; // Entry iterator
	MinArrayIndex				: DINT; // Minimum index of TU Array
	MaxArrayIndex				: DINT; // Maximum index of TU Array
	StartIndex					: DINT; // Start index of current iteration
	EndIndex					: DINT; // End index of current iteration
	IterationCounter			: DINT; // Iteration counter
	FoundOnBranch				: BOOL; // Checkpoint ID found on one of the configured branches
	BranchRecursive				: BOOL := TRUE; // Recursive branch search active (Default = True)
	

	CurrentNextTU_Index			: DINT; // Current next TU Index
	State						: INT; // State machine, 0=Idle, 1 = Search
	fbTrigExecute				: R_TRIG; // Trigger new request
	
	LowestNextSequence			: ULINT; // Lowest possible next sequence number
	LowestNextSubSequence		: DINT; // Lowest possible next sub sequence number
	rTU_DataEntry				: REFERENCE TO ST_TU_Data; // Currently checked entry
END_VAR

// Monitor new request trigger
fbTrigExecute(CLK := Execute);

CASE State OF
	// Idle - State
	0:
		// Wait for new start trigger
		IF fbTrigExecute.Q THEN
			// Validate inputs
			IF Sequence = 0 OR
			   Destination.eFunctionNumber = E_FunctionNumber.F_BEGIN_FUNCTION OR
			   Branch = 0 THEN
			   // Invalid inputs
			   Error := TRUE;
			   RETURN;
			END_IF
			
			// Initialize 
			Error := FALSE;
			Busy := TRUE;

			IterationCounter := 0;
			NextTU_Index := 0;
			NextTU_Checkpoint := '';
			CurrentNextTU_Index := 0;
			LowestNextSequence := 0;
			LowestNextSubSequence := 0;
			
			MinArrayIndex := 1; //LOWER_BOUND(TU_Table,1);
			MaxArrayIndex := Conveyor.NUMBER_OF_TU_DATA; //UPPER_BOUND(TU_Table,1);
			State := 1;
		END_IF
		
	// Iterate over multiple cycles through TU Table	
	1:
		StartIndex := MinArrayIndex + IterationCounter * EntriesPerCycle;
		EndIndex   := StartIndex + EntriesPerCycle;
	
		FOR EntryIdx := StartIndex TO EndIndex DO
			// When scan of TU is complete
			IF EntryIdx > MaxArrayIndex THEN
				// No possible next found
				IF CurrentNextTU_Index = 0 THEN
					NextTU_Index := 0;
					NextTU_Checkpoint := '';
					
				// Otherwise, ensure found index is still valid
				ELSE
					IF M_IsFoundNextIndexValid(TU_Table) THEN
						NextTU_Index := CurrentNextTU_Index;
						NextTU_Checkpoint := TU_Table[NextTU_Index].DataSet.CheckpointID;
						
					ELSE
						NextTU_Index := 0;
						NextTU_Checkpoint := '';
						
						Error := TRUE;
					END_IF
				END_IF
				
				Busy := FALSE;
			
				State := 0;
				RETURN;
			END_IF
			
			rTU_DataEntry REF= TU_Table[EntryIdx];
			
			// Skip this loop if...
            // - own index is found
            // - Empty data set is found
			// - Data set without job present is found ( no destination)
			IF EntryIdx = TU_Index OR 
               NOT rTU_DataEntry.DataSet.DataPresent OR 
               NOT rTU_DataEntry.DataSet.JobPresent THEN
				CONTINUE;
			END_IF
			
			// Check if TU has same Destination and Destination slot, 
			// otherwise it is not relevant for sequencing of requesting TU
			IF rTU_DataEntry.Destination[1].eFunctionNumber = Destination.eFunctionNumber AND
			   rTU_DataEntry.Destination[1].ZoneNumber = Destination.ZoneNumber THEN
				IF rTU_DataEntry.DataSet.DestinationSlot = DestinationSlot THEN
					
					// TU's can be ignored if...
					// - Sequence is lower than requesting sequence
					// - Sequence is 0 and is therefore not part of a sequence
					// - Sequence is higher than an already found next sequence
					// - Sequence is equal to requesting, but subsequence is lower
					IF rTU_DataEntry.DataSet.Sequence < Sequence OR
					   rTU_DataEntry.DataSet.Sequence = 0 OR
					   (rTU_DataEntry.DataSet.Sequence = Sequence AND
					   rTU_DataEntry.DataSet.SubSequence < SubSequence) OR   
					   (rTU_DataEntry.DataSet.Sequence > LowestNextSequence AND
					   LowestNextSequence <> 0) THEN
						// Skip
						;
				
					// Sequence is in a valid range for a possible next
					ELSE
						// check possible next TU
						IF rTU_DataEntry.DataSet.Sequence = LowestNextSequence THEN
							// Only lower sub sequences are checked for blocking
							IF rTU_DataEntry.DataSet.SubSequence < LowestNextSubSequence THEN
								// Check if current comapared TU is a possible next
								IF M_IsTU_Next(rTU_DataEntry) THEN
									LowestNextSubSequence := rTU_DataEntry.DataSet.SubSequence;
									
								   	// Store index and position at time when it was found
								   	CurrentNextTU_Index := EntryIdx;	
									
								// Otherwise the found TU is not influence sequencing of requesting
								ELSE
								   // Skip
								   ;
								END_IF
							END_IF
						// Less or equal
						ELSE
							// Check if current comapared TU is a possible next
							IF M_IsTU_Next(rTU_DataEntry) THEN
							   // TU is possible next, update Lowest next sequence pair
							   LowestNextSequence := rTU_DataEntry.DataSet.Sequence;
							   LowestNextSubSequence := rTU_DataEntry.DataSet.SubSequence;
							   
							   // Store index and position at time when it was found
							   CurrentNextTU_Index := EntryIdx;		
							END_IF
						END_IF
					END_IF
				END_IF
			END_IF
		END_FOR

		IterationCounter := IterationCounter + 1;
ELSE
	// Default
	State := 0;
END_CASE

/// This method checks if found index is still valid after a search over multiple cycles, 
/// because during search the state of index could have changed (Race condition).
METHOD PROTECTED M_IsFoundNextIndexValid : BOOL // Returns true if still valid, otherwise false
VAR_IN_OUT
	mTU_Table					: ARRAY[0..Conveyor.NUMBER_OF_TU_DATA] OF ST_TU_Data; // TU Table
END_VAR
VAR
	mrTU_DataEntry			: REFERENCE TO ST_TU_Data; // Currently checked entry
END_VAR
VAR_INST
	SequenceDataPresent		: BOOL; // Sequence data present
	TU_IsPartOfDestSequence	: BOOL; // Sequence data are for requested destination
END_VAR
M_IsFoundNextIndexValid := FALSE;

// Validate inputs
IF CurrentNextTU_Index <= 0 THEN
	RETURN;
END_IF

mrTU_DataEntry REF= mTU_Table[CurrentNextTU_Index];

// Check reference is valid
IF NOT __ISVALIDREF(mrTU_DataEntry) THEN
	RETURN;
END_IF

// Validate its TU data
// - Sequencing, 
// - Part of that sequence (destination)
// - Still at the detected checkpoint
SequenceDataPresent := mrTU_DataEntry.DataSet.Sequence > 0 AND
					   mrTU_DataEntry.Destination[1].eFunctionNumber > 0;
					   
TU_IsPartOfDestSequence := mrTU_DataEntry.Destination[1].eFunctionNumber = Destination.eFunctionNumber AND
						   mrTU_DataEntry.Destination[1].ZoneNumber = Destination.ZoneNumber AND
						   mrTU_DataEntry.DataSet.DestinationSlot = DestinationSlot;

IF SequenceDataPresent AND
   TU_IsPartOfDestSequence THEN	

	M_IsFoundNextIndexValid := M_IsTU_Next(rTU_DataEntry);
END_IF
END_METHOD

/// Check if current comapared TU is:
/// - Not located,
/// - Found on branch (Default mode) or Not found on a branch (Exclusion mode) 
/// Sequencing is temporarily haltet for this TU				
/// so its a possible next TU
METHOD PROTECTED M_IsTU_Next : BOOL // Returns true if it is a possible next
VAR_INPUT
	mrTU_DataEntry		: REFERENCE TO ST_TU_Data; // Currently checked entry
END_VAR
VAR
	mFoundOnBranch		: BOOL;
END_VAR
M_IsTU_Next := FALSE;

// Ensure it is still a problem for the branch	
mFoundOnBranch := Branch.M_IsOnBranches(BranchRecursive, mrTU_DataEntry.DataSet.CheckpointID);

IF (mFoundOnBranch AND NOT BranchExclusionMode) OR
   (NOT mFoundOnBranch AND BranchExclusionMode) OR
   (mrTU_DataEntry.DataSet.CheckpointID = '') OR
    mrTU_DataEntry.DataSet.HaltSequencing THEN
   
   M_IsTU_Next := TRUE;
END_IF
END_METHOD

{attribute 'monitoring' := 'call'}
/// Recursive branch search active. Remark: No automated loop detection.
PROPERTY P_BranchRecursive : BOOL
GET
P_BranchRecursive := BranchRecursive;
END_GET
SET
BranchRecursive := P_BranchRecursive;
END_SET
END_PROPERTY

/// TU Entries scanned per cycle
PROPERTY P_EntriesPerCycle : DINT // Default 600
GET
P_EntriesPerCycle := EntriesPerCycle;
END_GET
SET
EntriesPerCycle := P_EntriesPerCycle;
END_SET
END_PROPERTY

END_FUNCTION_BLOCK

// ---- 20_Product/30_Toolbox/16_Sequencing/10_Core/FB_SeqLimitedStream.TcPOU
/// Functionblock to maintain a specialized sequence-stream. 
FUNCTION_BLOCK FB_SeqLimitedStream
VAR_OUTPUT
	List: ARRAY[1..LIST_SIZE] OF DINT; // List of all TU indices
	EntryCounter: INT; // Counter of  entries in table
END_VAR
VAR CONSTANT
	LIST_SIZE: INT:= SequencingParameter.MAX_LIMITED_STREAM_LIST; // Size of limited stream
END_VAR

;

/// Add single TU index to list
METHOD M_Add : BOOL // True = TU index added, otherwise false
VAR_INPUT
	mTU_Index	: DINT;
END_VAR
VAR_IN_OUT
	mTU_Table	: ARRAY[0..Conveyor.NUMBER_OF_TU_DATA] OF ST_TU_Data; 	/// TU Table
END_VAR
VAR
	mIdx		: INT;
END_VAR
M_Add := FALSE;

// Validate input
IF mTU_Index> 0 AND mTU_Index< Conveyor.NUMBER_OF_TU_DATA THEN
	FOR mIdx := 1 TO LIST_SIZE DO
 	// Ensure data slot is free 
		IF List[mIdx] = 0  THEN
			List[mIdx] := mTU_Index;
			EntryCounter := EntryCounter + 1;
			mTU_Table[mTU_Index].DataSet.HaltSequencing := TRUE; // Mark TU as "Special Sequencing"
			M_Add := TRUE;
			RETURN;
			
		// TU Idx already registered
		ELSIF List[mIdx] = mTU_Index THEN
			mTU_Table[mTU_Index].DataSet.HaltSequencing := TRUE; // Mark TU as "Special Sequencing"
			M_Add := TRUE;
			RETURN;
			
		END_IF
	END_FOR
END_IF
END_METHOD

/// Removes a TU index from the list
METHOD M_Remove : BOOL // True = TU index removed , otherwise false
VAR_INPUT
	mTU_Index		: DINT; // TU index to remove
END_VAR
VAR_IN_OUT
	mTU_Table		: ARRAY[0..Conveyor.NUMBER_OF_TU_DATA] OF ST_TU_Data; // TU Table
END_VAR
VAR
	mIdx			: INT;
	mRemovedIdx		: INT;
	mSizeOneSlot	: UDINT;
END_VAR
M_Remove := TRUE;

// Validate inputs
IF mTU_Index <= 0 OR mTU_Index > Conveyor.NUMBER_OF_TU_DATA THEN
	M_Remove := FALSE;
	RETURN;
END_IF

// Search  object in table
FOR mIdx := 1 TO EntryCounter DO
	// Compare Element
	IF List[mIdx] = mTU_Index THEN

		// Unmark in TU table
		mTU_Table[List[mIdx]].DataSet.HaltSequencing := FALSE;
	
		// Clear slot 
		List[mIdx]:=0;	
		mRemovedIdx := mIdx;	
				
		// Update list and close gaps 
		// Shift subsequent entries
		IF mRemovedIdx < EntryCounter THEN
			mSizeOneSlot:= SIZEOF(List[1]);
			MEMCPY(ADR(List[mRemovedIdx]), ADR(List[mRemovedIdx+1]), INT_TO_UDINT(EntryCounter - mRemovedIdx) * mSizeOneSlot);
			List[EntryCounter]:=0;	
		END_IF
		
		EntryCounter := EntryCounter - 1;
	
		// Check counter border
		IF EntryCounter < 0 THEN
			EntryCounter := 0;
		END_IF
		EXIT;
	END_IF	
END_FOR
END_METHOD

/// Deletes all list entries
METHOD M_Clear : BOOL // True = All list entries deleted, otherwise false
VAR_IN_OUT
	mTU_Table	: ARRAY[0..Conveyor.NUMBER_OF_TU_DATA] OF ST_TU_Data; // TU Table
END_VAR
VAR
	mIdx		: INT;
END_VAR

FOR mIdx:= 1 TO EntryCounter DO
	// Unmark in TU table
	mTU_Table[mIdx].DataSet.HaltSequencing := FALSE;
	
END_FOR

// Update counter
EntryCounter := 0;

// Clear internal list
M_Clear := MEMSET(ADR(List), 0, SIZEOF(List)) > 0;
END_METHOD

/// Add multiple TU indices to the list at once
METHOD M_AddMultiple : BOOL // True =  All TU indeces added, otherwise false
VAR_IN_OUT
	mTU_Index		 : ARRAY [*] OF DINT; // Array of TU indices
END_VAR
VAR_IN_OUT
	mTU_Table		: ARRAY[0..Conveyor.NUMBER_OF_TU_DATA] OF ST_TU_Data; 	// TU Table
END_VAR
VAR
	mUpperBound		: DINT;
	mLowerBound		: DINT;
	mIdx			: DINT;
	mTU_Added		: BOOL;
END_VAR
// Assign lower and upper bound of input array
mLowerBound:= LOWER_BOUND(mTU_Index, 1);
mUpperBound:= UPPER_BOUND(mTU_Index, 1);
mTU_Added:= FALSE;

FOR mIdx:= mLowerBound TO mUpperBound DO
	// Add index to list, when input index is valid
	IF mTU_Index[mIdx]> 0 AND mTU_Index[mIdx]< Conveyor.NUMBER_OF_TU_DATA THEN
		mTU_Added:= mTU_Added AND M_Add(mTU_Index[mIdx], mTU_Table);		
	END_IF
END_FOR

M_AddMultiple:= mTU_Added;
END_METHOD

/// Checks if the requesting TU is blocked by a TU registered in the table. 
METHOD M_RequestRelease : BOOL // True =  Movement released, False = TU is beeing blocked
VAR_INPUT
	mTU_Index				: DINT; // Requesting TU Index
	mBranch					: I_BranchCheckpoint; // Branch to check
END_VAR
VAR_IN_OUT
	mTU_Table				: ARRAY[0..Conveyor.NUMBER_OF_TU_DATA] OF ST_TU_Data; // TU Table
END_VAR
VAR
	mIdx					: DINT;
	mLowestBlockingTU		: ST_TU_Data;
	mFoundOnBranch			: BOOL; /// False = TU on a branch is possible next, TRUE = TU on a branch is excluded as possible next
	mBranchExclusionMode	: BOOL := FALSE;
	mBranchRecursive		: BOOL := TRUE; // Recursive branch search active (Default = True)
	mRequestingTU_Present	: BOOL;
	mRequestingTU_Data		: ST_TU_Data;
	mListTU_Data			: ST_TU_Data;
END_VAR
VAR_OUTPUT
	mError					: BOOL; // True when inputs are invalid
END_VAR
M_RequestRelease:=FALSE;

// Validate input branch and TU index
IF mBranch = 0 OR
	 mTU_Index <= 0 OR mTU_Index > Conveyor.NUMBER_OF_TU_DATA THEN	
	mError:= TRUE;
	RETURN;
END_IF

// Get TU data from requesting index
mRequestingTU_Data:= mTU_Table[mTU_Index];

// 	Return when requesting TU is not in the list (not marked)
IF 	mRequestingTU_Data.DataSet.HaltSequencing = FALSE THEN	
	RETURN;
END_IF


// Find blocking TU on branch
//****************************************************************************
mLowestBlockingTU:= mRequestingTU_Data;


FOR mIdx:= 1 TO EntryCounter DO
	// Get TU data from list entry
	mListTU_Data:= mTU_Table[List[mIdx]];	
	
	// Only consider TU's which have the same destination and destination slot as the requesting one
	IF mRequestingTU_Data.Destination[1].eFunctionNumber = mListTU_Data.Destination[1].eFunctionNumber  AND
		mRequestingTU_Data.Destination[1].ZoneNumber = mListTU_Data.Destination[1].ZoneNumber AND
			mRequestingTU_Data.DataSet.DestinationSlot = mListTU_Data.DataSet.DestinationSlot THEN	
	
		// TU's can be ignored if...
		// - Sequence is 0 and is therefore not part of a sequence
		// - Sequence is equal to requesting, but subsequence is higher
		// - Sequence is higher than an already found lower sequence
		
		IF  mListTU_Data.DataSet.Sequence = 0 OR
		   (mListTU_Data.DataSet.Sequence = mLowestBlockingTU.DataSet.Sequence AND
			mListTU_Data.DataSet.SubSequence > mLowestBlockingTU.DataSet.SubSequence) OR
		   (mListTU_Data.DataSet.Sequence  > mLowestBlockingTU.DataSet.Sequence) THEN

			;// Skip
		
		// Possible Blocking TU 
		ELSE
			
			// When Sequence is the same the subsequence has to be checked additionally
			IF mListTU_Data.DataSet.Sequence = mLowestBlockingTU.DataSet.Sequence THEN
				
				// Only lower sub sequences are checked for blocking
				IF mListTU_Data.DataSet.SubSequence < mLowestBlockingTU.DataSet.SubSequence THEN
			
					mFoundOnBranch:= mBranch.M_IsOnBranches(mRecursive:= mBranchRecursive, mListTU_Data.DataSet.CheckpointID);
					
					IF ((mFoundOnBranch > 0 AND NOT mBranchExclusionMode) OR
						(mFoundOnBranch = 0 AND mBranchExclusionMode)) THEN
					
						mLowestBlockingTU:= mListTU_Data;		
					END_IF	
				END_IF
			
			ELSE // Sequence number is lower than last found blocking sequence
	
					mFoundOnBranch:= mBranch.M_IsOnBranches(mRecursive:= mBranchRecursive, mListTU_Data.DataSet.CheckpointID);
					
					IF ((mFoundOnBranch > 0 AND NOT mBranchExclusionMode) OR
						(mFoundOnBranch = 0 AND mBranchExclusionMode)) THEN
					
						mLowestBlockingTU:= mListTU_Data;		
					END_IF	
				
			END_IF	
		END_IF
	END_IF
END_FOR

 // Dont release if blocking TU is found and its not the requesting TU
IF mLowestBlockingTU.TU_ID.HashCode > 0 AND
	 mLowestBlockingTU.TU_ID.HashCode <> mRequestingTU_Data.TU_ID.HashCode  THEN
	 
	 M_RequestRelease:=FALSE;
	 
ELSE 
	 M_RequestRelease:=TRUE;
END_IF
END_METHOD

END_FUNCTION_BLOCK

// ---- 20_Product/30_Toolbox/16_Sequencing/10_Core/F_UpdateCheckpointID.TcPOU
/// Updates checkpoint ID of TU data slot
FUNCTION F_UpdateCheckpointID : BOOL // True if update was successful
(************************************************************************************** 
* 	Application 		: BoxControl Framework 
* 	Revision 			: $Revision: 404877 $ 
* 	Revision date 		: $Date: 2018-04-26 14:10:34 +0200 (Thu, 26 Apr 2018) $ 
* 	Last changed by 	: $Author: b7ernsb $ 
* 	URL 				: $URL: http://almscdc.swisslog.com/repo/SWPD/Development/BoxControlFramework/21_Projects/BCF_2.0/trunk/BCF/BCF/JumpStart/20_Product/10_App/12_E_Functions/10_Lib/10_Conv/FB_FunctionConv.TcPOU $ 
* ------------------------------------------------------------------------------------ 
* 	© Swisslog AG 
* 	Swisslog is not liable for any usage of this source code that is not agreed 
* 	on between Swisslog and the other party. The mandatory legal liability remains 
* 	unaffected. 
* ------------------------------------------------------------------------------------ 
* 	Revision History: 
* 
* 	VERSION 		DATE 			INITIALS 			DESCRIPTION 
* 	0.1 			23.05.2018 		mbo 				Created.
* 
**************************************************************************************)
VAR_INPUT
	Enable		: BOOL; // Enable update
	CheckpointID: STRING(5); // Checkpoint ID to update
END_VAR
VAR_IN_OUT
	TU_Data		: ST_TU_Data; // TU data set to be updated
END_VAR

F_UpdateCheckpointID := FALSE;

IF Enable THEN
	TU_Data.DataSet.CheckpointID := CheckpointID;
	F_UpdateCheckpointID := TRUE;

END_IF

END_FUNCTION

// ---- 20_Product/30_Toolbox/16_Sequencing/11_Strategies/FB_SeqCheckpoint.TcPOU
/// Checkpoint updates all passing TUs and can be used
/// as part of a sequencing tree-
FUNCTION_BLOCK FB_SeqCheckpoint IMPLEMENTS I_BranchCheckpoint
(************************************************************************************** 
* 	Application 		: BoxControl Framework 
* 	Revision 			: $Revision: 404877 $ 
* 	Revision date 		: $Date: 2018-04-26 14:10:34 +0200 (Thu, 26 Apr 2018) $ 
* 	Last changed by 	: $Author: b7ernsb $ 
* 	URL 				: $URL: http://almscdc.swisslog.com/repo/SWPD/Development/BoxControlFramework/21_Projects/BCF_2.0/trunk/BCF/BCF/JumpStart/20_Product/10_App/12_E_Functions/10_Lib/10_Conv/FB_FunctionConv.TcPOU $ 
* ------------------------------------------------------------------------------------ 
* 	© Swisslog AG 
* 	Swisslog is not liable for any usage of this source code that is not agreed 
* 	on between Swisslog and the other party. The mandatory legal liability remains 
* 	unaffected. 
* ------------------------------------------------------------------------------------ 
* 	Revision History: 
* 
* 	VERSION 		DATE 			INITIALS 			DESCRIPTION 
* 	0.1 			23.05.2018 		mbo 				Created.
* 
**************************************************************************************)
VAR_INPUT
	Enable		: BOOL; // Enable checkpoint update
	CheckpointID: STRING(5); // Checkpoint id to update
END_VAR
VAR_IN_OUT
	TU_Data		: ST_TU_Data; // Tu data set
END_VAR


IF Enable THEN
	TU_Data.DataSet.CheckpointID := CheckpointID;
END_IF

/// Identifier for checkpoint
{attribute 'monitoring' := 'call'}
{attribute 'suppress_wrn_C0410'}
PROPERTY P_CheckpointID : REFERENCE TO STRING(5)
GET
P_CheckpointID REF= CheckpointID;
END_GET
END_PROPERTY

/// Searches if a checkpoint can be found on a specific branch
METHOD M_IsOnBranches : BOOL // Returns true if found, false = not found 
VAR_INPUT
	mRecursive	: BOOL := FALSE; // Search recursive through the whole tree
END_VAR
VAR_IN_OUT CONSTANT
	mCheckpointID	: STRING(5); // Last checkpoint id	
END_VAR

M_IsOnBranches := mCheckpointID = P_CheckpointID;
END_METHOD

END_FUNCTION_BLOCK

// ---- 20_Product/30_Toolbox/16_Sequencing/11_Strategies/FB_SeqEstimateAllNextTUs.TcPOU
/// Estimates next TU after the requesting one. Does the same as FB_SeqEstimateNextTU
/// but can handle multiple destination streams.
FUNCTION_BLOCK FB_SeqEstimateAllNextTUs IMPLEMENTS I_SeqEstimateNext
(************************************************************************************** 
* 	Application 		: BoxControl Framework 
* 	Revision 			: $Revision: 404877 $ 
* 	Revision date 		: $Date: 2018-04-26 14:10:34 +0200 (Thu, 26 Apr 2018) $ 
* 	Last changed by 	: $Author: b7ernsb $ 
* 	URL 				: $URL: http://almscdc.swisslog.com/repo/SWPD/Development/BoxControlFramework/21_Projects/BCF_2.0/trunk/BCF/BCF/JumpStart/20_Product/10_App/12_E_Functions/10_Lib/10_Conv/FB_FunctionConv.TcPOU $ 
* ------------------------------------------------------------------------------------ 
* 	© Swisslog AG 
* 	Swisslog is not liable for any usage of this source code that is not agreed 
* 	on between Swisslog and the other party. The mandatory legal liability remains 
* 	unaffected. 
* ------------------------------------------------------------------------------------ 
* 	Revision History: 
* 
* 	VERSION 		DATE 			INITIALS 			DESCRIPTION 
* 	0.1 			23.05.2018 		mbo 				Created.
*	0.2				08.02.2019		mbo					Racecondition fixed
* 
**************************************************************************************)
VAR_INPUT
	Execute					: BOOL; // Requires rising edge for new request
	TU_Present				: BOOL; // A TU is present on branch A
	TU_Index				: DINT; // Waiting TU data index A
	Branch					: I_BranchCheckpoint; // Branch to check for next branch
	BranchExclusionMode		: BOOL := FALSE; // False = TU on a branch is possible next, TRUE = TU on a branch is excluded as possible next
END_VAR
VAR_OUTPUT
	Busy					: BOOL; // Process ongoing
	Error					: BOOL; // Error during process (configuration error)
	NextTU_List				: ARRAY[1..MAX_LIST_ENTRIES] OF ST_SeqEntry; // List of next expected TUs for all passing sequences
	ListCount				: INT; // Available entries in list
END_VAR
VAR_IN_OUT
	TU_Table				: ARRAY[0..Conveyor.NUMBER_OF_TU_DATA] OF ST_TU_Data; // TU Table
END_VAR
VAR
	State					: INT; // State machine 0: Request 1: Search
	fbTrigExecute			: R_TRIG; // Trigger new request
	SequenceDataPresent 	: BOOL; // Sequence data available
	RequestedDestination	: ST_PositionIdent; // Requested destination for search
	RequestedDestinationSlot: INT; // Requested destination slot for search
	fbSeqGetNextTU			: FB_SeqGetNextTU; // Get next following TU of this sequence
	NextTU_Index			: DINT;
END_VAR
VAR CONSTANT
	MAX_LIST_ENTRIES		: INT := SequencingParameter.MAX_ESTIMATE_ALL_NEXT_LIST;
END_VAR

// Monitor new request trigger
fbTrigExecute(CLK := Execute);

CASE State OF
	// Wait for a new TU
	0:
		// Wait for new start trigger
		IF fbTrigExecute.Q THEN
			// Validate inputs
			IF Branch = 0 THEN
				Error := TRUE;
				RETURN;
			END_IF
			
			// Process started...
			Busy := TRUE;
			Error := FALSE;
			NextTU_Index := 0;
			RequestedDestination.eFunctionNumber := E_FunctionNumber.F_BEGIN_FUNCTION;
			RequestedDestination.ZoneNumber := 0;

			// When a requesting TU is present
			IF TU_Present THEN

				IF TU_Index > 0 THEN
					// If the TU consists of sequencing information
					SequenceDataPresent := TU_Table[TU_Index].DataSet.Sequence > 0 AND
					                       TU_Table[TU_Index].Destination[1].eFunctionNumber > 0;
										   
					IF SequenceDataPresent  THEN
						// Store destination to valid after search
						RequestedDestination := TU_Table[TU_Index].Destination[1];
						RequestedDestinationSlot := TU_Table[TU_Index].DataSet.DestinationSlot;
						
